C03656=1147.991,39.631,-50.274,-179.877,6.308,149.107
C03657=1147.986,39.881,-50.290,-179.875,6.309,149.107
C03658=1147.981,40.130,-50.305,-179.871,6.310,149.106
C03659=1147.976,40.380,-50.321,-179.869,6.311,149.106
C03660=1147.971,40.630,-50.335,-179.866,6.312,149.105
C03661=1147.966,40.879,-50.350,-179.864,6.313,149.105
C03662=1147.961,41.128,-50.365,-179.861,6.315,149.104
C03663=1147.956,41.378,-50.381,-179.859,6.315,149.104
C03664=1147.951,41.627,-50.395,-179.856,6.316,149.103
C03665=1147.945,41.877,-50.411,-179.853,6.317,149.102
C03666=1147.941,42.126,-50.426,-179.851,6.318,149.102
C03667=1147.936,42.376,-50.442,-179.848,6.320,149.102
C03668=1147.931,42.626,-50.456,-179.846,6.320,149.101
C03669=1147.926,42.875,-50.472,-179.843,6.322,149.100
C03670=1147.921,43.124,-50.487,-179.840,6.323,149.100
C03671=1147.916,43.374,-50.502,-179.838,6.323,149.099
C03672=1147.910,43.623,-50.518,-179.835,6.325,149.099
C03673=1147.906,43.872,-50.533,-179.833,6.325,149.098
C03674=1147.901,44.122,-50.549,-179.830,6.327,149.098
C03675=1147.896,44.372,-50.563,-179.827,6.328,149.097
C03676=1147.890,44.621,-50.579,-179.824,6.329,149.097
C03677=1147.885,44.871,-50.594,-179.822,6.330,149.096
C03678=1147.880,45.120,-50.609,-179.819,6.331,149.096
C03679=1147.876,45.370,-50.625,-179.817,6.332,149.095
C03680=1147.870,45.619,-50.641,-179.814,6.333,149.094
C03681=1147.866,45.868,-50.656,-179.812,6.334,149.094
C03682=1147.860,46.118,-50.671,-179.809,6.335,149.094
C03683=1147.856,46.367,-50.686,-179.806,6.336,149.093
C03684=1147.851,46.617,-50.702,-179.804,6.337,149.092
C03685=1147.845,46.866,-50.718,-179.801,6.339,149.092
C03686=1147.841,47.115,-50.733,-179.799,6.339,149.091
C03687=1147.835,47.365,-50.748,-179.796,6.341,149.091
C03688=1147.831,47.615,-50.764,-179.793,6.342,149.090
C03689=1147.826,47.864,-50.779,-179.790,6.343,149.090
C03690=1147.821,48.113,-50.795,-179.788,6.344,149.089
C03691=1147.815,48.363,-50.811,-179.785,6.345,149.089
C03692=1147.810,48.613,-50.827,-179.783,6.346,149.088
C03693=1147.806,48.862,-50.842,-179.780,6.347,149.088
C03694=1147.800,49.111,-50.857,-179.777,6.348,149.087
C03695=1147.795,49.361,-50.873,-179.775,6.349,149.087
C03696=1147.791,49.611,-50.888,-179.772,6.350,149.086
C03697=1147.785,49.860,-50.904,-179.770,6.351,149.086
C03698=1147.780,50.109,-50.919,-179.767,6.352,149.085
C03699=1147.775,50.359,-50.935,-179.765,6.353,149.084
C03700=1147.771,50.609,-50.950,-179.762,6.355,149.084
C03701=1147.765,50.858,-50.966,-179.759,6.355,149.083
C03702=1147.760,51.107,-50.982,-179.756,6.357,149.083
C03703=1147.755,51.357,-50.998,-179.754,6.358,149.082
C03704=1147.750,51.606,-51.014,-179.751,6.359,149.082
C03705=1147.745,51.855,-51.029,-179.749,6.360,149.081
C03706=1147.741,52.105,-51.045,-179.746,6.361,149.081
C03707=1147.735,52.355,-51.060,-179.743,6.362,149.080
C03708=1147.730,52.604,-51.076,-179.741,6.364,149.080
C03709=1147.725,52.854,-51.092,-179.738,6.364,149.079
C03710=1147.721,53.103,-51.107,-179.735,6.366,149.079
C03711=1147.715,53.371,-51.124,-179.732,6.367,149.078
C03712=1147.710,53.640,-51.141,-179.730,6.368,149.078
C03713=1147.704,53.908,-51.158,-179.727,6.369,149.077
C03714=1147.699,54.177,-51.176,-179.724,6.371,149.076
C03715=1147.694,54.427,-51.191,-179.721,6.371,149.076
C03716=1147.688,54.676,-51.207,-179.719,6.373,149.075
C03717=1147.684,54.926,-51.224,-179.716,6.374,149.075
C03718=1147.678,55.175,-51.239,-179.713,6.375,149.074
C03719=1147.673,55.425,-51.255,-179.711,6.376,149.074
C03720=1147.669,55.674,-51.270,-179.708,6.378,149.073
C03721=1147.664,55.923,-51.287,-179.706,6.378,149.073
C03722=1147.659,56.173,-51.302,-179.703,6.380,149.072
C03723=1147.654,56.423,-51.318,-179.700,6.380,149.072
C03724=1147.649,56.671,-51.334,-179.697,6.382,149.071
C03725=1147.644,56.922,-51.350,-179.695,6.383,149.071
C03726=1147.638,57.171,-51.366,-179.692,6.384,149.070
C03727=1147.633,57.420,-51.382,-179.689,6.386,149.070
C03728=1147.629,57.670,-51.398,-179.687,6.387,149.069
C03729=1147.624,57.919,-51.414,-179.684,6.388,149.068
C03730=1147.619,58.169,-51.430,-179.682,6.389,149.068
C03731=1147.613,58.418,-51.446,-179.679,6.390,149.068
C03732=1147.609,58.668,-51.463,-179.676,6.391,149.067
C03733=1147.603,58.917,-51.478,-179.674,6.393,149.067
C03734=1147.598,59.166,-51.495,-179.671,6.393,149.066
C03735=1147.594,59.416,-51.511,-179.668,6.395,149.065
C03736=1147.589,59.665,-51.527,-179.666,6.396,149.065
C03737=1147.584,59.915,-51.543,-179.663,6.397,149.064
C03738=1147.579,60.164,-51.559,-179.660,6.399,149.064
C03739=1147.574,60.414,-51.575,-179.658,6.399,149.063
C03740=1147.569,60.662,-51.591,-179.655,6.401,149.063
C03741=1147.564,60.913,-51.607,-179.653,6.402,149.062
C03742=1147.559,61.161,-51.624,-179.650,6.403,149.062
C03743=1147.554,61.411,-51.640,-179.647,6.404,149.061
C03744=1147.549,61.660,-51.656,-179.644,6.405,149.061
C03745=1147.544,61.910,-51.672,-179.642,6.406,149.060
C03746=1147.539,62.159,-51.688,-179.639,6.407,149.060
C03747=1147.534,62.409,-51.704,-179.636,6.409,149.059
C03748=1147.529,62.658,-51.720,-179.634,6.410,149.059
C03749=1147.524,62.908,-51.738,-179.631,6.411,149.058
C03750=1147.519,63.157,-51.753,-179.629,6.412,149.058
C03751=1147.514,63.407,-51.770,-179.626,6.414,149.057
C03752=1147.509,63.656,-51.785,-179.623,6.414,149.057
C03753=1147.504,63.906,-51.802,-179.621,6.416,149.056
C03754=1147.499,64.154,-51.818,-179.618,6.418,149.056
C03755=1147.495,64.404,-51.834,-179.615,6.418,149.055
C03756=1147.489,64.653,-51.851,-179.613,6.420,149.055
C03757=1147.484,64.903,-51.868,-179.610,6.420,149.054
C03758=1147.479,65.152,-51.884,-179.607,6.422,149.054
C03759=1147.474,65.402,-51.900,-179.604,6.424,149.053
C03760=1147.469,65.651,-51.917,-179.602,6.424,149.052
C03761=1147.464,65.901,-51.933,-179.599,6.426,149.052
C03762=1147.460,66.150,-51.949,-179.597,6.427,149.052
C03763=1147.454,66.399,-51.966,-179.594,6.428,149.051
C03764=1147.450,66.649,-51.983,-179.591,6.429,149.050
C03765=1147.444,66.898,-51.998,-179.589,6.430,149.050
C03766=1147.440,67.148,-52.015,-179.586,6.432,149.049
C03767=1147.435,67.397,-52.031,-179.583,6.432,149.049
C03768=1147.430,67.646,-52.049,-179.581,6.434,149.049
C03769=1147.425,67.896,-52.065,-179.577,6.435,149.048
C03770=1147.420,68.145,-52.081,-179.575,6.436,149.047
C03771=1147.415,68.395,-52.097,-179.572,6.438,149.047
C03772=1147.409,68.644,-52.114,-179.570,6.439,149.047
C03773=1147.405,68.893,-52.131,-179.567,6.440,149.046
C03774=1147.400,69.143,-52.148,-179.564,6.442,149.045
C03775=1147.395,69.392,-52.163,-179.562,6.443,149.045
C03776=1147.390,69.642,-52.181,-179.559,6.444,149.044
C03777=1147.385,69.891,-52.197,-179.556,6.446,149.044
C03778=1147.380,70.140,-52.214,-179.554,6.446,149.044
C03779=1147.375,70.390,-52.231,-179.551,6.448,149.043
C03780=1147.371,70.640,-52.247,-179.549,6.449,149.042
C03781=1147.365,70.888,-52.264,-179.546,6.450,149.042
C03782=1147.361,71.138,-52.280,-179.543,6.452,149.041
C03783=1147.355,71.387,-52.297,-179.541,6.452,149.041
C03784=1147.350,71.637,-52.313,-179.538,6.454,149.040
C03785=1147.346,71.886,-52.330,-179.535,6.455,149.040
C03786=1147.340,72.136,-52.347,-179.532,6.456,149.039
C03787=1147.336,72.385,-52.364,-179.530,6.458,149.039
C03788=1147.330,72.635,-52.381,-179.527,6.459,149.038
C03789=1147.326,72.884,-52.397,-179.524,6.460,149.038
C03790=1147.321,73.133,-52.414,-179.522,6.462,149.037
C03791=1147.316,73.383,-52.431,-179.519,6.463,149.037
C03792=1147.311,73.632,-52.448,-179.516,6.464,149.036
C03793=1147.306,73.881,-52.464,-179.514,6.466,149.036
C03794=1147.301,74.131,-52.481,-179.511,6.466,149.035
C03795=1147.296,74.380,-52.498,-179.508,6.468,149.035
C03796=1147.291,74.629,-52.516,-179.505,6.469,149.034
C03797=1147.286,74.878,-52.532,-179.503,6.470,149.034
C03798=1147.281,75.128,-52.550,-179.500,6.472,149.033
C03799=1147.277,75.378,-52.566,-179.497,6.473,149.033
C03800=1147.272,75.626,-52.582,-179.495,6.474,149.032
C03801=1147.266,75.876,-52.600,-179.492,6.475,149.032
C03802=1147.262,76.126,-52.616,-179.489,6.477,149.031
C03803=1147.257,76.376,-52.634,-179.487,6.478,149.031
C03804=1147.252,76.624,-52.650,-179.484,6.480,149.031
C03805=1147.246,76.874,-52.667,-179.481,6.481,149.030
C03806=1147.242,77.123,-52.685,-179.479,6.482,149.029
C03807=1147.237,77.373,-52.702,-179.476,6.483,149.029
C03808=1147.232,77.622,-52.718,-179.473,6.485,149.028
C03809=1147.227,77.871,-52.735,-179.471,6.486,149.028
C03810=1147.222,78.121,-52.752,-179.468,6.487,149.027
C03811=1147.217,78.370,-52.770,-179.465,6.489,149.027
C03812=1147.213,78.620,-52.787,-179.462,6.490,149.026
C03813=1147.207,78.869,-52.804,-179.460,6.491,149.026
C03814=1147.202,79.118,-52.821,-179.457,6.493,149.026
C03815=1147.197,79.387,-52.839,-179.454,6.494,149.025
C03816=1147.191,79.654,-52.858,-179.451,6.496,149.024
C03817=1147.187,79.923,-52.876,-179.448,6.497,149.024
C03818=1147.181,80.192,-52.895,-179.446,6.498,149.023
C03819=1147.176,80.441,-52.912,-179.443,6.499,149.023
C03820=1147.171,80.691,-52.928,-179.440,6.501,149.022
C03821=1147.166,80.940,-52.946,-179.437,6.502,149.022
C03822=1147.162,81.189,-52.963,-179.435,6.503,149.021
C03823=1147.156,81.439,-52.980,-179.432,6.505,149.021
C03824=1147.152,81.688,-52.998,-179.429,6.506,149.020
C03825=1147.147,81.938,-53.015,-179.427,6.507,149.020
C03826=1147.141,82.187,-53.032,-179.424,6.509,149.020
C03827=1147.136,82.436,-53.050,-179.421,6.510,149.019
C03828=1147.132,82.685,-53.067,-179.418,6.512,149.018
C03829=1147.127,82.935,-53.085,-179.416,6.513,149.018
C03830=1147.122,83.184,-53.102,-179.413,6.514,149.018
C03831=1147.117,83.434,-53.118,-179.410,6.516,149.017
C03832=1147.112,83.683,-53.136,-179.408,6.517,149.017
C03833=1147.107,83.933,-53.154,-179.405,6.518,149.016
C03834=1147.102,84.181,-53.171,-179.402,6.520,149.016
C03835=1147.097,84.431,-53.188,-179.399,6.521,149.015
C03836=1147.092,84.680,-53.206,-179.397,6.522,149.015
C03837=1147.088,84.929,-53.223,-179.394,6.524,149.014
C03838=1147.083,85.179,-53.241,-179.391,6.525,149.014
C03839=1147.078,85.428,-53.258,-179.388,6.527,149.013
C03840=1147.073,85.678,-53.276,-179.386,6.528,149.013
C03841=1147.068,85.927,-53.293,-179.384,6.529,149.012
C03842=1147.063,86.176,-53.311,-179.380,6.531,149.012
C03843=1147.058,86.426,-53.328,-179.378,6.532,149.011
C03844=1147.053,86.675,-53.346,-179.375,6.533,149.011
C03845=1147.049,86.925,-53.362,-179.373,6.535,149.010
C03846=1147.044,87.174,-53.380,-179.369,6.536,149.010
C03847=1147.038,87.422,-53.398,-179.367,6.538,149.009
C03848=1147.033,87.672,-53.415,-179.365,6.539,149.009
C03849=1147.028,87.921,-53.433,-179.362,6.540,149.008
C03850=1147.024,88.171,-53.450,-179.359,6.542,149.008
C03851=1147.019,88.420,-53.468,-179.356,6.543,149.007
C03852=1147.014,88.669,-53.486,-179.354,6.544,149.007
C03853=1147.009,88.919,-53.503,-179.351,6.546,149.007
C03854=1147.004,89.168,-53.521,-179.348,6.547,149.006
C03855=1147.000,89.417,-53.539,-179.345,6.549,149.005
C03856=1146.994,89.667,-53.556,-179.343,6.550,149.005
C03857=1146.989,89.916,-53.574,-179.340,6.551,149.005
C03858=1146.984,90.165,-53.592,-179.337,6.553,149.004
C03859=1146.979,90.415,-53.609,-179.334,6.554,149.004
C03860=1146.974,90.664,-53.627,-179.332,6.555,149.003
C03861=1146.969,90.913,-53.645,-179.329,6.557,149.003
C03862=1146.965,91.162,-53.663,-179.327,6.559,149.002
C03863=1146.960,91.412,-53.680,-179.323,6.560,149.002
C03864=1146.955,91.661,-53.698,-179.321,6.562,149.001
C03865=1146.951,91.911,-53.716,-179.319,6.562,149.001
C03866=1146.946,92.160,-53.734,-179.316,6.564,149.000
C03867=1146.941,92.410,-53.751,-179.313,6.565,149.000
C03868=1146.936,92.659,-53.769,-179.310,6.567,148.999
C03869=1146.931,92.908,-53.787,-179.308,6.568,148.999
C03870=1146.926,93.157,-53.805,-179.305,6.570,148.998
C03871=1146.921,93.407,-53.823,-179.302,6.571,148.998
C03872=1146.916,93.656,-53.840,-179.299,6.573,148.997
C03873=1146.911,93.906,-53.858,-179.296,6.574,148.997
C03874=1146.906,94.155,-53.876,-179.294,6.575,148.997
C03875=1146.901,94.404,-53.894,-179.291,6.577,148.996
C03876=1146.896,94.653,-53.912,-179.288,6.578,148.995
C03877=1146.891,94.902,-53.930,-179.285,6.580,148.995
C03878=1146.886,95.152,-53.948,-179.283,6.582,148.995
C03879=1146.882,95.401,-53.967,-179.281,6.582,148.994
C03880=1146.877,95.651,-53.985,-179.278,6.584,148.994
C03881=1146.872,95.900,-54.003,-179.275,6.585,148.993
C03882=1146.867,96.150,-54.020,-179.272,6.587,148.993
C03883=1146.862,96.399,-54.038,-179.269,6.589,148.992
C03884=1146.857,96.648,-54.056,-179.266,6.590,148.992
C03885=1146.852,96.897,-54.074,-179.264,6.591,148.991
C03886=1146.847,97.146,-54.092,-179.261,6.593,148.991
C03887=1146.843,97.396,-54.110,-179.258,6.594,148.990
C03888=1146.838,97.645,-54.128,-179.256,6.596,148.990
C03889=1146.833,97.894,-54.146,-179.253,6.598,148.990
C03890=1146.828,98.144,-54.164,-179.250,6.599,148.989
C03891=1146.823,98.393,-54.183,-179.248,6.600,148.989
C03892=1146.818,98.642,-54.201,-179.245,6.602,148.988
C03893=1146.814,98.892,-54.220,-179.242,6.603,148.988
C03894=1146.809,99.141,-54.238,-179.239,6.605,148.987
C03895=1146.804,99.390,-54.256,-179.237,6.607,148.987
C03896=1146.799,99.639,-54.274,-179.233,6.608,148.986
C03897=1146.794,99.888,-54.292,-179.231,6.609,148.986
C03898=1146.789,100.137,-54.310,-179.229,6.611,148.985
C03899=1146.784,100.388,-54.328,-179.226,6.612,148.985
C03900=1146.779,100.637,-54.346,-179.223,6.614,148.985
C03901=1146.774,100.886,-54.364,-179.220,6.615,148.984
C03902=1146.770,101.135,-54.383,-179.217,6.617,148.984
C03903=1146.765,101.384,-54.401,-179.215,6.618,148.983
C03904=1146.760,101.634,-54.419,-179.212,6.619,148.983
C03905=1146.755,101.883,-54.438,-179.210,6.621,148.982
C03906=1146.750,102.132,-54.456,-179.207,6.623,148.982
C03907=1146.745,102.381,-54.475,-179.204,6.624,148.981
C03908=1146.741,102.631,-54.493,-179.201,6.626,148.981
C03909=1146.735,102.880,-54.512,-179.198,6.628,148.980
C03910=1146.730,103.129,-54.530,-179.195,6.629,148.980
C03911=1146.726,103.378,-54.548,-179.193,6.630,148.980
C03912=1146.722,103.628,-54.567,-179.190,6.631,148.979
C03913=1146.716,103.877,-54.585,-179.187,6.633,148.979
C03914=1146.711,104.126,-54.603,-179.185,6.635,148.978
C03915=1146.707,104.376,-54.622,-179.182,6.636,148.978
C03916=1146.702,104.625,-54.640,-179.179,6.638,148.977
C03917=1146.696,104.874,-54.659,-179.176,6.640,148.977
C03918=1146.692,105.123,-54.678,-179.173,6.641,148.976
C03919=1146.687,105.392,-54.697,-179.170,6.643,148.976
C03920=1146.681,105.660,-54.717,-179.168,6.645,148.975
C03921=1146.676,105.929,-54.737,-179.165,6.646,148.975
C03922=1146.671,106.197,-54.757,-179.162,6.648,148.974
C03923=1146.667,106.447,-54.776,-179.159,6.649,148.974
C03924=1146.661,106.695,-54.795,-179.156,6.651,148.974
C03925=1146.656,106.945,-54.813,-179.154,6.653,148.973
C03926=1146.652,107.194,-54.831,-179.151,6.654,148.973
C03927=1146.647,107.443,-54.851,-179.148,6.655,148.972
C03928=1146.642,107.692,-54.869,-179.146,6.657,148.972
C03929=1146.638,107.942,-54.888,-179.143,6.658,148.971
C03930=1146.632,108.191,-54.906,-179.140,6.660,148.971
C03931=1146.628,108.440,-54.925,-179.137,6.662,148.970
C03932=1146.622,108.690,-54.944,-179.135,6.663,148.970
C03933=1146.618,108.939,-54.963,-179.132,6.665,148.970
C03934=1146.613,109.188,-54.981,-179.129,6.666,148.969
C03935=1146.608,109.437,-55.000,-179.126,6.668,148.969
C03936=1146.603,109.686,-55.018,-179.123,6.670,148.968
C03937=1146.598,109.935,-55.038,-179.121,6.671,148.968
C03938=1146.594,110.185,-55.056,-179.118,6.672,148.967
C03939=1146.588,110.434,-55.075,-179.116,6.674,148.967
C03940=1146.584,110.684,-55.094,-179.113,6.676,148.967
C03941=1146.579,110.933,-55.113,-179.110,6.677,148.966
C03942=1146.574,111.181,-55.132,-179.107,6.679,148.966
C03943=1146.569,111.432,-55.150,-179.104,6.680,148.965
C03944=1146.564,111.680,-55.169,-179.102,6.682,148.965
C03945=1146.559,111.930,-55.188,-179.099,6.684,148.964
C03946=1146.555,112.179,-55.207,-179.096,6.685,148.964
C03947=1146.550,112.428,-55.226,-179.093,6.687,148.963
C03948=1146.545,112.678,-55.244,-179.091,6.689,148.963
C03949=1146.540,112.926,-55.264,-179.087,6.690,148.962
C03950=1146.536,113.176,-55.283,-179.085,6.692,148.962
C03951=1146.530,113.425,-55.301,-179.082,6.693,148.962
C03952=1146.526,113.674,-55.320,-179.079,6.695,148.961
C03953=1146.521,113.923,-55.340,-179.077,6.696,148.961
C03954=1146.516,114.173,-55.358,-179.074,6.698,148.960
C03955=1146.511,114.422,-55.377,-179.072,6.699,148.960
C03956=1146.506,114.672,-55.397,-179.069,6.701,148.960
C03957=1146.502,114.920,-55.416,-179.066,6.703,148.959
C03958=1146.497,115.170,-55.435,-179.063,6.704,148.959
C03959=1146.492,115.419,-55.453,-179.060,6.706,148.958
C03960=1146.487,115.668,-55.473,-179.058,6.708,148.958
C03961=1146.482,115.917,-55.492,-179.055,6.709,148.957
C03962=1146.478,116.167,-55.511,-179.052,6.711,148.957
C03963=1146.472,116.416,-55.530,-179.049,6.713,148.957
C03964=1146.468,116.666,-55.550,-179.047,6.714,148.956
C03965=1146.463,116.914,-55.568,-179.044,6.716,148.956
C03966=1146.458,117.164,-55.588,-179.041,6.718,148.955
C03967=1146.453,117.413,-55.607,-179.038,6.719,148.955
C03968=1146.449,117.662,-55.626,-179.035,6.721,148.954
C03969=1146.444,117.911,-55.646,-179.033,6.722,148.954
C03970=1146.439,118.160,-55.665,-179.030,6.724,148.953
C03971=1146.434,118.410,-55.683,-179.027,6.726,148.953
C03972=1146.429,118.659,-55.703,-179.024,6.728,148.953
C03973=1146.424,118.908,-55.722,-179.022,6.729,148.952
C03974=1146.420,119.157,-55.741,-179.019,6.731,148.952
C03975=1146.415,119.407,-55.761,-179.016,6.733,148.951
C03976=1146.410,119.656,-55.780,-179.014,6.734,148.951
C03977=1146.405,119.905,-55.800,-179.011,6.736,148.951
C03978=1146.400,120.154,-55.818,-179.008,6.738,148.950
C03979=1146.396,120.403,-55.838,-179.005,6.739,148.950
C03980=1146.390,120.652,-55.857,-179.002,6.741,148.949
C03981=1146.386,120.902,-55.877,-178.999,6.742,148.949
C03982=1146.382,121.151,-55.896,-178.997,6.744,148.948
C03983=1146.376,121.400,-55.915,-178.994,6.746,148.948
C03984=1146.371,121.649,-55.935,-178.991,6.748,148.948
C03985=1146.366,121.898,-55.954,-178.989,6.749,148.947
C03986=1146.361,122.148,-55.974,-178.986,6.751,148.947
C03987=1146.357,122.397,-55.993,-178.983,6.753,148.946
C03988=1146.352,122.645,-56.013,-178.980,6.754,148.946
C03989=1146.348,122.895,-56.033,-178.978,6.756,148.946
C03990=1146.343,123.145,-56.052,-178.975,6.758,148.945
C03991=1146.337,123.393,-56.072,-178.972,6.759,148.945
C03992=1146.333,123.643,-56.091,-178.969,6.761,148.944
C03993=1146.329,123.892,-56.110,-178.967,6.763,148.944
C03994=1146.323,124.141,-56.130,-178.964,6.765,148.944
C03995=1146.319,124.390,-56.150,-178.961,6.766,148.943
C03996=1146.314,124.640,-56.170,-178.958,6.768,148.943
C03997=1146.309,124.889,-56.189,-178.955,6.769,148.942
C03998=1146.304,125.138,-56.209,-178.953,6.771,148.942
C03999=1146.299,125.388,-56.228,-178.950,6.773,148.941
C04000=1146.294,125.636,-56.248,-178.947,6.774,148.941
C04001=1146.290,125.885,-56.267,-178.945,6.776,148.941
C04002=1146.286,126.135,-56.287,-178.942,6.778,148.940
C04003=1146.280,126.384,-56.306,-178.939,6.780,148.940
C04004=1146.276,126.633,-56.327,-178.936,6.781,148.939
C04005=1146.271,126.882,-56.346,-178.934,6.783,148.939
C04006=1146.266,127.132,-56.366,-178.931,6.785,148.939
C04007=1146.261,127.380,-56.386,-178.928,6.786,148.938
C04008=1146.257,127.629,-56.406,-178.925,6.788,148.938
C04009=1146.252,127.879,-56.425,-178.922,6.791,148.937
C04010=1146.247,128.128,-56.446,-178.919,6.792,148.937
C04011=1146.242,128.377,-56.465,-178.917,6.794,148.937
C04012=1146.237,128.626,-56.485,-178.914,6.796,148.936
C04013=1146.233,128.875,-56.505,-178.911,6.797,148.936
C04014=1146.228,129.125,-56.525,-178.909,6.799,148.935
C04015=1146.223,129.374,-56.544,-178.906,6.801,148.935
C04016=1146.218,129.623,-56.564,-178.903,6.802,148.935
C04017=1146.214,129.872,-56.584,-178.900,6.804,148.934
C04018=1146.209,130.121,-56.604,-178.898,6.806,148.934
C04019=1146.204,130.370,-56.624,-178.895,6.808,148.933
C04020=1146.199,130.619,-56.644,-178.892,6.809,148.933
C04021=1146.195,130.869,-56.664,-178.890,6.811,148.933
C04022=1146.189,131.118,-56.685,-178.887,6.813,148.932
C04023=1146.185,131.387,-56.706,-178.884,6.815,148.932
C04024=1146.180,131.655,-56.727,-178.880,6.817,148.931
C04025=1146.174,131.924,-56.749,-178.878,6.818,148.931
C04026=1146.169,132.192,-56.770,-178.874,6.821,148.931
C04027=1146.164,132.441,-56.790,-178.872,6.822,148.930
C04028=1146.159,132.690,-56.811,-178.869,6.824,148.930
C04029=1146.154,132.939,-56.831,-178.866,6.826,148.929
C04030=1146.150,133.189,-56.851,-178.863,6.828,148.929
C04031=1146.145,133.438,-56.871,-178.861,6.829,148.929
C04032=1146.140,133.687,-56.891,-178.858,6.831,148.928
C04033=1146.136,133.936,-56.911,-178.855,6.833,148.928
C04034=1146.130,134.186,-56.931,-178.853,6.834,148.927
C04035=1146.125,134.434,-56.951,-178.849,6.837,148.927
C04036=1146.121,134.683,-56.972,-178.847,6.839,148.927
C04037=1146.116,134.933,-56.991,-178.844,6.840,148.926
C04038=1146.112,135.182,-57.012,-178.841,6.842,148.926
C04039=1146.107,135.431,-57.033,-178.838,6.844,148.925
C04040=1146.102,135.681,-57.052,-178.836,6.845,148.925
C04041=1146.098,135.930,-57.073,-178.833,6.847,148.925
C04042=1146.092,136.178,-57.093,-178.830,6.849,148.924
C04043=1146.088,136.427,-57.113,-178.828,6.851,148.924
C04044=1146.083,136.677,-57.133,-178.824,6.853,148.923
C04045=1146.078,136.926,-57.154,-178.822,6.855,148.923
C04046=1146.074,137.175,-57.174,-178.819,6.857,148.923
C04047=1146.069,137.424,-57.195,-178.816,6.858,148.922
C04048=1146.064,137.674,-57.215,-178.813,6.860,148.922
C04049=1146.059,137.922,-57.235,-178.811,6.862,148.922
C04050=1146.055,138.171,-57.255,-178.808,6.863,148.921
C04051=1146.050,138.421,-57.276,-178.805,6.866,148.921
C04052=1146.045,138.670,-57.297,-178.802,6.868,148.921
C04053=1146.041,138.919,-57.316,-178.800,6.870,148.920
C04054=1146.035,139.168,-57.337,-178.797,6.871,148.920
C04055=1146.031,139.417,-57.358,-178.794,6.873,148.919
C04056=1146.026,139.666,-57.378,-178.792,6.875,148.919
C04057=1146.021,139.916,-57.399,-178.789,6.876,148.919
C04058=1146.016,140.164,-57.419,-178.786,6.879,148.918
C04059=1146.012,140.413,-57.439,-178.783,6.881,148.918
C04060=1146.007,140.662,-57.460,-178.780,6.882,148.917
C04061=1146.002,140.912,-57.480,-178.777,6.884,148.917
C04062=1145.997,141.161,-57.501,-178.775,6.886,148.917
C04063=1145.992,141.410,-57.521,-178.772,6.888,148.916
C04064=1145.988,141.659,-57.542,-178.769,6.889,148.916
C04065=1145.983,141.909,-57.563,-178.766,6.892,148.916
C04066=1145.979,142.158,-57.584,-178.763,6.893,148.915
C04067=1145.974,142.407,-57.604,-178.761,6.895,148.915
C04068=1145.969,142.656,-57.625,-178.758,6.897,148.914
C04069=1145.965,142.905,-57.645,-178.756,6.899,148.914
C04070=1145.960,143.154,-57.666,-178.753,6.901,148.914
C04071=1145.955,143.403,-57.687,-178.750,6.903,148.913
C04072=1145.950,143.652,-57.708,-178.747,6.905,148.913
C04073=1145.946,143.901,-57.729,-178.744,6.907,148.913
C04074=1145.941,144.150,-57.750,-178.741,6.908,148.912
C04075=1145.936,144.399,-57.770,-178.739,6.910,148.912
C04076=1145.931,144.648,-57.791,-178.735,6.913,148.912
C04077=1145.927,144.897,-57.811,-178.733,6.914,148.911
C04078=1145.922,145.146,-57.832,-178.730,6.916,148.911
C04079=1145.917,145.395,-57.853,-178.727,6.918,148.910
C04080=1145.912,145.645,-57.874,-178.725,6.919,148.910
C04081=1145.907,145.893,-57.894,-178.722,6.922,148.910
C04082=1145.903,146.143,-57.916,-178.719,6.924,148.909
C04083=1145.899,146.392,-57.936,-178.716,6.926,148.909
C04084=1145.894,146.641,-57.957,-178.714,6.927,148.909
C04085=1145.888,146.890,-57.978,-178.711,6.929,148.908
C04086=1145.884,147.139,-57.999,-178.708,6.931,148.908
C04087=1145.879,147.388,-58.020,-178.705,6.933,148.908
C04088=1145.875,147.637,-58.041,-178.702,6.935,148.907
C04089=1145.869,147.886,-58.062,-178.699,6.937,148.907
C04090=1145.865,148.136,-58.083,-178.697,6.939,148.906
C04091=1145.861,148.384,-58.104,-178.695,6.941,148.906
C04092=1145.856,148.634,-58.125,-178.691,6.943,148.906
C04093=1145.851,148.883,-58.145,-178.689,6.945,148.905
C04094=1145.846,149.131,-58.167,-178.686,6.947,148.905
C04095=1145.841,149.380,-58.188,-178.683,6.948,148.905
C04096=1145.837,149.629,-58.209,-178.680,6.951,148.904
C04097=1145.832,149.879,-58.230,-178.677,6.953,148.904
C04098=1145.827,150.128,-58.252,-178.674,6.954,148.904
C04099=1145.823,150.377,-58.272,-178.672,6.956,148.903
C04100=1145.818,150.626,-58.294,-178.669,6.958,148.903
C04101=1145.813,150.875,-58.315,-178.666,6.961,148.903
C04102=1145.808,151.125,-58.336,-178.663,6.962,148.902
C04103=1145.804,151.373,-58.357,-178.661,6.964,148.902
C04104=1145.799,151.622,-58.378,-178.658,6.966,148.901
C04105=1145.794,151.871,-58.400,-178.655,6.968,148.901
C04106=1145.790,152.120,-58.420,-178.652,6.970,148.901
C04107=1145.785,152.369,-58.442,-178.650,6.972,148.901
C04108=1145.780,152.619,-58.463,-178.647,6.974,148.900
C04109=1145.775,152.868,-58.484,-178.644,6.976,148.900
C04110=1145.770,153.117,-58.506,-178.641,6.978,148.899
C04111=1145.766,153.366,-58.526,-178.638,6.980,148.899
C04112=1145.761,153.615,-58.548,-178.636,6.981,148.899
C04113=1145.757,153.863,-58.570,-178.632,6.984,148.898
C04114=1145.751,154.113,-58.591,-178.630,6.986,148.898
C04115=1145.747,154.362,-58.613,-178.627,6.988,148.898
C04116=1145.743,154.611,-58.633,-178.625,6.990,148.897
C04117=1145.738,154.860,-58.655,-178.621,6.992,148.897
C04118=1145.733,155.109,-58.676,-178.619,6.994,148.897
C04119=1145.728,155.358,-58.698,-178.616,6.995,148.896
C04120=1145.723,155.607,-58.720,-178.614,6.998,148.896
C04121=1145.718,155.856,-58.740,-178.610,7.000,148.896
C04122=1145.715,156.105,-58.762,-178.608,7.002,148.895
C04123=1145.710,156.354,-58.783,-178.605,7.004,148.895
C04124=1145.705,156.603,-58.805,-178.602,7.006,148.895
C04125=1145.700,156.852,-58.826,-178.599,7.008,148.894
C04126=1145.695,157.102,-58.848,-178.597,7.010,148.894
C04127=1145.691,157.370,-58.871,-178.594,7.012,148.894
C04128=1145.685,157.639,-58.894,-178.591,7.014,148.893
C04129=1145.681,157.909,-58.917,-178.588,7.017,148.893
C04130=1145.675,158.177,-58.941,-178.585,7.018,148.893
C04131=1145.670,158.427,-58.962,-178.582,7.021,148.892
C04132=1145.665,158.675,-58.984,-178.579,7.023,148.892
C04133=1145.661,158.924,-59.006,-178.576,7.024,148.892
C04134=1145.656,159.173,-59.028,-178.574,7.026,148.891
C04135=1145.651,159.422,-59.049,-178.571,7.029,148.891
C04136=1145.647,159.672,-59.071,-178.568,7.031,148.891
C04137=1145.642,159.920,-59.092,-178.565,7.032,148.890
C04138=1145.637,160.169,-59.114,-178.562,7.035,148.890
C04139=1145.633,160.418,-59.136,-178.560,7.037,148.890
C04140=1145.628,160.667,-59.158,-178.557,7.039,148.889
C04141=1145.624,160.916,-59.180,-178.554,7.041,148.889
C04142=1145.618,161.166,-59.201,-178.551,7.043,148.889
C04143=1145.614,161.414,-59.222,-178.548,7.045,148.888
C04144=1145.609,161.664,-59.245,-178.545,7.048,148.888
C04145=1145.604,161.912,-59.266,-178.543,7.049,148.888
C04146=1145.600,162.162,-59.288,-178.540,7.051,148.887
C04147=1145.595,162.410,-59.310,-178.537,7.054,148.887
C04148=1145.591,162.660,-59.332,-178.534,7.055,148.887
C04149=1145.586,162.908,-59.354,-178.532,7.057,148.886
C04150=1145.581,163.157,-59.375,-178.529,7.059,148.886
C04151=1145.577,163.406,-59.397,-178.526,7.062,148.886
C04152=1145.572,163.655,-59.419,-178.523,7.063,148.885
C04153=1145.568,163.904,-59.441,-178.521,7.065,148.885
C04154=1145.562,164.153,-59.463,-178.518,7.068,148.885
C04155=1145.558,164.402,-59.485,-178.515,7.070,148.884
C04156=1145.553,164.651,-59.507,-178.512,7.071,148.884
C04157=1145.549,164.900,-59.529,-178.509,7.074,148.884
C04158=1145.544,165.149,-59.551,-178.507,7.076,148.884
C04159=1145.540,165.398,-59.573,-178.503,7.079,148.883
C04160=1145.535,165.647,-59.595,-178.501,7.080,148.883
C04161=1145.530,165.897,-59.617,-178.498,7.082,148.883
C04162=1145.525,166.145,-59.639,-178.495,7.085,148.882
C04163=1145.521,166.394,-59.662,-178.492,7.087,148.882
C04164=1145.516,166.643,-59.683,-178.490,7.088,148.882
C04165=1145.512,166.892,-59.705,-178.487,7.091,148.881
C04166=1145.506,167.141,-59.728,-178.484,7.093,148.881
C04167=1145.502,167.390,-59.750,-178.482,7.095,148.881
C04168=1145.497,167.639,-59.771,-178.478,7.097,148.880
C04169=1145.493,167.888,-59.794,-178.476,7.099,148.880
C04170=1145.488,168.137,-59.816,-178.473,7.101,148.880
C04171=1145.483,168.386,-59.839,-178.470,7.104,148.880
C04172=1145.479,168.635,-59.861,-178.467,7.105,148.879
C04173=1145.474,168.884,-59.882,-178.464,7.108,148.879
C04174=1145.469,169.133,-59.906,-178.462,7.110,148.879
C04175=1145.465,169.382,-59.927,-178.459,7.112,148.878
C04176=1145.460,169.631,-59.949,-178.456,7.114,148.878
C04177=1145.455,169.879,-59.972,-178.454,7.116,148.878
C04178=1145.451,170.129,-59.994,-178.451,7.118,148.877
C04179=1145.447,170.378,-60.016,-178.448,7.121,148.877
C04180=1145.441,170.626,-60.039,-178.445,7.123,148.877
C04181=1145.437,170.876,-60.061,-178.442,7.125,148.877
C04182=1145.432,171.124,-60.083,-178.439,7.127,148.876
C04183=1145.427,171.373,-60.106,-178.437,7.129,148.876
C04184=1145.423,171.623,-60.129,-178.434,7.132,148.876
C04185=1145.418,171.871,-60.150,-178.431,7.133,148.875
C04186=1145.414,172.120,-60.174,-178.428,7.136,148.875
C04187=1145.409,172.369,-60.195,-178.426,7.138,148.875
C04188=1145.404,172.618,-60.219,-178.423,7.140,148.874
C04189=1145.400,172.867,-60.241,-178.420,7.142,148.874
C04190=1145.395,173.116,-60.262,-178.417,7.144,148.874
C04191=1145.390,173.365,-60.286,-178.414,7.147,148.874
C04192=1145.386,173.614,-60.308,-178.411,7.149,148.873
C04193=1145.381,173.863,-60.331,-178.409,7.151,148.873
C04194=1145.376,174.112,-60.353,-178.406,7.153,148.873
C04195=1145.372,174.361,-60.376,-178.403,7.155,148.872
C04196=1145.367,174.610,-60.398,-178.400,7.157,148.872
C04197=1145.362,174.859,-60.421,-178.398,7.160,148.872
C04198=1145.358,175.107,-60.444,-178.395,7.161,148.871
C04199=1145.354,175.357,-60.466,-178.392,7.164,148.871
C04200=1145.349,175.605,-60.489,-178.390,7.166,148.871
C04201=1145.344,175.854,-60.511,-178.386,7.168,148.871
C04202=1145.340,176.104,-60.534,-178.384,7.170,148.870
C04203=1145.335,176.352,-60.556,-178.381,7.173,148.870
C04204=1145.330,176.601,-60.579,-178.378,7.175,148.870
C04205=1145.325,176.850,-60.603,-178.375,7.177,148.869
C04206=1145.321,177.100,-60.625,-178.373,7.179,148.869
C04207=1145.316,177.348,-60.648,-178.370,7.181,148.869
C04208=1145.312,177.597,-60.671,-178.367,7.184,148.869
C04209=1145.307,177.846,-60.693,-178.364,7.186,148.868
C04210=1145.303,178.095,-60.716,-178.361,7.188,148.868
C04211=1145.297,178.343,-60.739,-178.359,7.190,148.868
C04212=1145.294,178.592,-60.762,-178.356,7.193,148.868
C04213=1145.289,178.842,-60.784,-178.353,7.195,148.867
C04214=1145.284,179.091,-60.808,-178.351,7.197,148.867
C04215=1145.279,179.339,-60.830,-178.347,7.199,148.867
C04216=1145.275,179.588,-60.854,-178.345,7.201,148.866
C04217=1145.270,179.837,-60.876,-178.342,7.204,148.866
C04218=1145.266,180.086,-60.899,-178.339,7.206,148.866
C04219=1145.261,180.335,-60.922,-178.336,7.208,148.866
C04220=1145.256,180.583,-60.945,-178.334,7.210,148.865
C04221=1145.252,180.832,-60.968,-178.330,7.213,148.865
C04222=1145.247,181.082,-60.991,-178.328,7.215,148.865
C04223=1145.243,181.331,-61.013,-178.325,7.218,148.865
C04224=1145.238,181.580,-61.037,-178.322,7.219,148.864
C04225=1145.233,181.829,-61.060,-178.319,7.222,148.864
C04226=1145.229,182.077,-61.083,-178.317,7.224,148.864
C04227=1145.224,182.326,-61.106,-178.313,7.226,148.863
C04228=1145.219,182.575,-61.129,-178.311,7.229,148.863
C04229=1145.215,182.824,-61.153,-178.308,7.230,148.863
C04230=1145.211,183.073,-61.175,-178.306,7.233,148.863
C04231=1145.205,183.342,-61.200,-178.302,7.236,148.862
C04232=1145.200,183.612,-61.226,-178.299,7.238,148.862
C04233=1145.195,183.882,-61.251,-178.296,7.240,148.862
C04234=1145.190,184.151,-61.275,-178.294,7.243,148.862
C04235=1145.185,184.400,-61.298,-178.290,7.245,148.861
C04236=1145.181,184.649,-61.322,-178.288,7.248,148.861
C04237=1145.176,184.898,-61.346,-178.285,7.250,148.861
C04238=1145.172,185.147,-61.369,-178.282,7.252,148.860
C04239=1145.168,185.395,-61.392,-178.279,7.255,148.860
C04240=1145.163,185.645,-61.415,-178.277,7.256,148.860
C04241=1145.158,185.894,-61.439,-178.274,7.259,148.860
C04242=1145.154,186.143,-61.462,-178.271,7.261,148.859
C04243=1145.148,186.391,-61.485,-178.268,7.264,148.859
C04244=1145.144,186.640,-61.508,-178.266,7.266,148.859
C04245=1145.140,186.889,-61.531,-178.262,7.268,148.859
C04246=1145.135,187.138,-61.554,-178.260,7.270,148.859
C04247=1145.130,187.387,-61.578,-178.257,7.273,148.858
C04248=1145.126,187.635,-61.602,-178.255,7.275,148.858
C04249=1145.121,187.884,-61.625,-178.251,7.278,148.858
C04250=1145.116,188.133,-61.649,-178.249,7.280,148.858
C04251=1145.112,188.382,-61.672,-178.246,7.282,148.857
C04252=1145.107,188.631,-61.695,-178.243,7.284,148.857
C04253=1145.103,188.880,-61.719,-178.240,7.287,148.857
C04254=1145.098,189.129,-61.743,-178.238,7.289,148.856
C04255=1145.093,189.378,-61.766,-178.235,7.291,148.856
C04256=1145.088,189.627,-61.789,-178.232,7.293,148.856
C04257=1145.085,189.875,-61.813,-178.229,7.296,148.856
C04258=1145.080,190.124,-61.836,-178.227,7.298,148.855
C04259=1145.075,190.373,-61.860,-178.224,7.301,148.855
C04260=1145.071,190.621,-61.884,-178.221,7.303,148.855
C04261=1145.066,190.870,-61.907,-178.218,7.305,148.855
C04262=1145.062,191.119,-61.930,-178.215,7.308,148.855
C04263=1145.057,191.368,-61.955,-178.212,7.310,148.854
C04264=1145.052,191.617,-61.978,-178.210,7.313,148.854
C04265=1145.047,191.866,-62.002,-178.207,7.314,148.854
C04266=1145.043,192.115,-62.026,-178.204,7.317,148.854
C04267=1145.038,192.364,-62.049,-178.201,7.319,148.853
C04268=1145.034,192.612,-62.073,-178.199,7.322,148.853
C04269=1145.029,192.861,-62.097,-178.195,7.324,148.853
C04270=1145.024,193.110,-62.120,-178.193,7.327,148.853
C04271=1145.020,193.359,-62.144,-178.190,7.329,148.852
C04272=1145.015,193.608,-62.167,-178.188,7.331,148.852
C04273=1145.011,193.857,-62.192,-178.184,7.334,148.852
C04274=1145.007,194.106,-62.215,-178.182,7.336,148.852
C04275=1145.002,194.354,-62.239,-178.179,7.338,148.851
C04276=1144.998,194.603,-62.263,-178.176,7.341,148.851
C04277=1144.992,194.852,-62.287,-178.173,7.343,148.851
C04278=1144.988,195.101,-62.311,-178.170,7.346,148.851
C04279=1144.983,195.349,-62.335,-178.168,7.348,148.850
C04280=1144.979,195.598,-62.359,-178.165,7.351,148.850
C04281=1144.974,195.847,-62.382,-178.162,7.352,148.850
C04282=1144.970,196.096,-62.407,-178.159,7.355,148.850
C04283=1144.965,196.345,-62.431,-178.156,7.358,148.850
C04284=1144.961,196.594,-62.455,-178.154,7.360,148.849
C04285=1144.956,196.842,-62.479,-178.151,7.362,148.849
C04286=1144.951,197.091,-62.502,-178.148,7.365,148.849
C04287=1144.947,197.340,-62.526,-178.145,7.367,148.849
C04288=1144.942,197.588,-62.551,-178.142,7.370,148.848
C04289=1144.938,197.838,-62.575,-178.140,7.372,148.848
C04290=1144.933,198.086,-62.599,-178.137,7.375,148.848
C04291=1144.929,198.335,-62.623,-178.135,7.377,148.848
C04292=1144.924,198.584,-62.647,-178.131,7.379,148.848
C04293=1144.919,198.833,-62.671,-178.129,7.382,148.847
C04294=1144.915,199.082,-62.695,-178.126,7.384,148.847
C04295=1144.911,199.330,-62.719,-178.123,7.387,148.847
C04296=1144.906,199.579,-62.743,-178.120,7.389,148.847
C04297=1144.901,199.828,-62.767,-178.118,7.391,148.847
C04298=1144.897,200.076,-62.791,-178.114,7.394,148.846
C04299=1144.892,200.326,-62.816,-178.112,7.396,148.846
C04300=1144.888,200.574,-62.841,-178.109,7.399,148.846
C04301=1144.883,200.823,-62.864,-178.107,7.401,148.846
C04302=1144.879,201.072,-62.888,-178.104,7.404,148.845
C04303=1144.874,201.321,-62.913,-178.101,7.406,148.845
C04304=1144.870,201.569,-62.937,-178.098,7.408,148.845
C04305=1144.865,201.818,-62.962,-178.095,7.411,148.845
C04306=1144.860,202.066,-62.986,-178.092,7.414,148.845
C04307=1144.857,202.316,-63.010,-178.090,7.416,148.844
C04308=1144.851,202.564,-63.035,-178.087,7.418,148.844
C04309=1144.847,202.813,-63.059,-178.084,7.421,148.844
C04310=1144.842,203.062,-63.082,-178.081,7.423,148.844
C04311=1144.838,203.311,-63.107,-178.078,7.426,148.844
C04312=1144.833,203.560,-63.131,-178.076,7.428,148.843
C04313=1144.828,203.808,-63.156,-178.073,7.431,148.843
C04314=1144.824,204.057,-63.181,-178.070,7.434,148.843
C04315=1144.819,204.306,-63.205,-178.067,7.435,148.843
C04316=1144.815,204.555,-63.229,-178.065,7.438,148.843
C04317=1144.810,204.804,-63.254,-178.061,7.441,148.842
C04318=1144.806,205.052,-63.279,-178.059,7.443,148.842
C04319=1144.802,205.300,-63.303,-178.056,7.446,148.842
C04320=1144.797,205.550,-63.328,-178.053,7.448,148.842
C04321=1144.792,205.798,-63.353,-178.051,7.450,148.842
C04322=1144.788,206.047,-63.377,-178.048,7.453,148.841
C04323=1144.783,206.296,-63.402,-178.045,7.456,148.841
C04324=1144.779,206.545,-63.426,-178.043,7.458,148.841
C04325=1144.774,206.793,-63.451,-178.039,7.461,148.841
C04326=1144.770,207.042,-63.475,-178.037,7.463,148.841
C04327=1144.765,207.291,-63.500,-178.034,7.466,148.840
C04328=1144.761,207.539,-63.525,-178.031,7.468,148.840
C04329=1144.756,207.788,-63.550,-178.028,7.471,148.840
C04330=1144.752,208.037,-63.574,-178.026,7.473,148.840
C04331=1144.747,208.286,-63.599,-178.023,7.476,148.840
C04332=1144.742,208.535,-63.624,-178.020,7.479,148.839
C04333=1144.738,208.783,-63.648,-178.017,7.480,148.839
C04334=1144.734,209.032,-63.673,-178.014,7.483,148.839
C04335=1144.728,209.302,-63.700,-178.012,7.486,148.839
C04336=1144.724,209.573,-63.727,-178.008,7.489,148.839
C04337=1144.719,209.843,-63.754,-178.006,7.492,148.839
C04338=1144.714,210.114,-63.781,-178.002,7.494,148.838
C04339=1144.709,210.363,-63.806,-178.000,7.497,148.838
C04340=1144.705,210.612,-63.831,-177.997,7.500,148.838
C04341=1144.700,210.860,-63.855,-177.994,7.502,148.838
C04342=1144.696,211.110,-63.880,-177.991,7.505,148.838
C04343=1144.691,211.358,-63.906,-177.988,7.508,148.837
C04344=1144.687,211.607,-63.930,-177.986,7.509,148.837
C04345=1144.682,211.855,-63.956,-177.983,7.512,148.837
C04346=1144.677,212.104,-63.980,-177.980,7.515,148.837
C04347=1144.673,212.353,-64.005,-177.977,7.518,148.837
C04348=1144.669,212.601,-64.030,-177.975,7.520,148.836
C04349=1144.664,212.850,-64.055,-177.972,7.523,148.836
C04350=1144.659,213.098,-64.081,-177.969,7.525,148.836
C04351=1144.655,213.348,-64.106,-177.966,7.527,148.836
C04352=1144.651,213.596,-64.130,-177.964,7.530,148.836
C04353=1144.646,213.845,-64.155,-177.960,7.533,148.836
C04354=1144.641,214.093,-64.181,-177.958,7.536,148.835
C04355=1144.637,214.343,-64.206,-177.955,7.538,148.835
C04356=1144.633,214.591,-64.231,-177.952,7.540,148.835
C04357=1144.628,214.840,-64.256,-177.949,7.543,148.835
C04358=1144.624,215.089,-64.281,-177.946,7.546,148.835
C04359=1144.619,215.337,-64.306,-177.944,7.548,148.835
C04360=1144.615,215.586,-64.332,-177.941,7.551,148.834
C04361=1144.610,215.834,-64.357,-177.938,7.554,148.834
C04362=1144.606,216.083,-64.382,-177.935,7.557,148.834
C04363=1144.601,216.331,-64.407,-177.933,7.559,148.834
C04364=1144.597,216.580,-64.433,-177.930,7.561,148.834
C04365=1144.592,216.830,-64.458,-177.927,7.564,148.834
C04366=1144.588,217.078,-64.483,-177.924,7.567,148.834
C04367=1144.583,217.327,-64.509,-177.922,7.569,148.833
C04368=1144.578,217.575,-64.534,-177.919,7.572,148.833
C04369=1144.574,217.824,-64.559,-177.916,7.575,148.833
C04370=1144.571,218.073,-64.585,-177.913,7.578,148.833
C04371=1144.565,218.321,-64.609,-177.911,7.580,148.833
C04372=1144.561,218.570,-64.635,-177.908,7.582,148.832
C04373=1144.556,218.818,-64.660,-177.905,7.585,148.832
C04374=1144.552,219.067,-64.686,-177.902,7.588,148.832
C04375=1144.548,219.316,-64.712,-177.899,7.590,148.832
C04376=1144.543,219.565,-64.737,-177.897,7.593,148.832
C04377=1144.539,219.813,-64.762,-177.894,7.596,148.832
C04378=1144.534,220.062,-64.788,-177.891,7.599,148.832
C04379=1144.530,220.310,-64.813,-177.888,7.601,148.831
C04380=1144.525,220.559,-64.839,-177.886,7.603,148.831
C04381=1144.521,220.808,-64.865,-177.883,7.606,148.831
C04382=1144.516,221.057,-64.890,-177.880,7.609,148.831
C04383=1144.512,221.305,-64.915,-177.877,7.612,148.831
C04384=1144.508,221.554,-64.941,-177.875,7.614,148.831
C04385=1144.503,221.802,-64.966,-177.872,7.617,148.831
C04386=1144.498,222.051,-64.992,-177.869,7.620,148.830
C04387=1144.494,222.300,-65.018,-177.866,7.622,148.830
C04388=1144.489,222.548,-65.043,-177.863,7.625,148.830
C04389=1144.484,222.797,-65.070,-177.861,7.627,148.830
C04390=1144.480,223.046,-65.095,-177.858,7.630,148.830
C04391=1144.475,223.294,-65.121,-177.855,7.633,148.830
C04392=1144.471,223.543,-65.147,-177.852,7.636,148.829
C04393=1144.467,223.792,-65.172,-177.849,7.639,148.829
C04394=1144.463,224.041,-65.198,-177.847,7.641,148.829
C04395=1144.458,224.289,-65.223,-177.844,7.644,148.829
C04396=1144.454,224.537,-65.249,-177.841,7.647,148.829
C04397=1144.449,224.786,-65.275,-177.838,7.649,148.829
C04398=1144.444,225.035,-65.301,-177.835,7.652,148.829
C04399=1144.440,225.283,-65.327,-177.833,7.654,148.828
C04400=1144.436,225.532,-65.353,-177.830,7.657,148.828
C04401=1144.432,225.780,-65.379,-177.827,7.660,148.828
C04402=1144.427,226.029,-65.405,-177.824,7.663,148.828
C04403=1144.422,226.278,-65.431,-177.821,7.666,148.828
C04404=1144.417,226.526,-65.456,-177.818,7.668,148.828
C04405=1144.413,226.775,-65.482,-177.816,7.671,148.828
C04406=1144.409,227.024,-65.508,-177.813,7.673,148.828
C04407=1144.405,227.272,-65.534,-177.810,7.676,148.827
C04408=1144.400,227.521,-65.560,-177.807,7.679,148.827
C04409=1144.395,227.769,-65.586,-177.805,7.682,148.827
C04410=1144.391,228.018,-65.612,-177.802,7.685,148.827
C04411=1144.386,228.267,-65.639,-177.800,7.687,148.827
C04412=1144.382,228.516,-65.665,-177.797,7.690,148.827
C04413=1144.377,228.764,-65.690,-177.794,7.692,148.827
C04414=1144.373,229.012,-65.717,-177.791,7.695,148.826
C04415=1144.369,229.261,-65.743,-177.788,7.698,148.826
C04416=1144.364,229.510,-65.769,-177.785,7.701,148.826
C04417=1144.360,229.759,-65.794,-177.783,7.703,148.826
C04418=1144.355,230.007,-65.821,-177.780,7.706,148.826
C04419=1144.351,230.256,-65.847,-177.777,7.709,148.826
C04420=1144.347,230.503,-65.873,-177.774,7.712,148.826
C04421=1144.342,230.752,-65.900,-177.771,7.715,148.826
C04422=1144.337,231.001,-65.925,-177.769,7.717,148.826
C04423=1144.334,231.249,-65.952,-177.766,7.720,148.825
C04424=1144.329,231.499,-65.978,-177.764,7.722,148.825
C04425=1144.325,231.747,-66.005,-177.761,7.725,148.825
C04426=1144.320,231.996,-66.031,-177.758,7.728,148.825
C04427=1144.316,232.244,-66.057,-177.755,7.731,148.825
C04428=1144.312,232.493,-66.083,-177.752,7.734,148.825
C04429=1144.306,232.741,-66.110,-177.749,7.737,148.825
C04430=1144.302,232.989,-66.136,-177.746,7.740,148.825
C04431=1144.297,233.238,-66.163,-177.743,7.743,148.825
C04432=1144.293,233.487,-66.188,-177.741,7.745,148.824
C04433=1144.289,233.735,-66.216,-177.738,7.748,148.824
C04434=1144.284,233.984,-66.241,-177.736,7.751,148.824
C04435=1144.280,234.233,-66.268,-177.733,7.753,148.824
C04436=1144.275,234.481,-66.294,-177.730,7.756,148.824
C04437=1144.271,234.730,-66.321,-177.727,7.759,148.824
C04438=1144.267,234.978,-66.348,-177.724,7.762,148.824
C04439=1144.261,235.250,-66.376,-177.721,7.765,148.824
C04440=1144.257,235.522,-66.405,-177.718,7.768,148.824
C04441=1144.253,235.794,-66.435,-177.716,7.771,148.823
C04442=1144.247,236.066,-66.463,-177.712,7.774,148.823
C04443=1144.243,236.314,-66.490,-177.709,7.777,148.823
C04444=1144.239,236.563,-66.517,-177.706,7.780,148.823
C04445=1144.234,236.811,-66.544,-177.704,7.782,148.823
C04446=1144.230,237.060,-66.570,-177.701,7.785,148.823
C04447=1144.225,237.309,-66.597,-177.698,7.788,148.823
C04448=1144.221,237.557,-66.623,-177.696,7.791,148.823
C04449=1144.216,237.805,-66.650,-177.693,7.794,148.823
C04450=1144.211,238.054,-66.677,-177.690,7.797,148.823
C04451=1144.208,238.303,-66.703,-177.687,7.799,148.822
C04452=1144.203,238.551,-66.730,-177.684,7.802,148.822
C04453=1144.199,238.799,-66.757,-177.682,7.805,148.822
C04454=1144.194,239.048,-66.784,-177.679,7.808,148.822
C04455=1144.189,239.297,-66.810,-177.676,7.811,148.822
C04456=1144.185,239.545,-66.837,-177.673,7.813,148.822
C04457=1144.181,239.793,-66.864,-177.671,7.816,148.822
C04458=1144.177,240.043,-66.891,-177.668,7.819,148.822
C04459=1144.173,240.291,-66.917,-177.665,7.822,148.822
C04460=1144.168,240.539,-66.945,-177.662,7.825,148.821
C04461=1144.163,240.788,-66.972,-177.659,7.827,148.821
C04462=1144.159,241.036,-66.999,-177.657,7.830,148.821
C04463=1144.155,241.285,-67.025,-177.654,7.833,148.821
C04464=1144.150,241.533,-67.052,-177.651,7.836,148.821
C04465=1144.146,241.782,-67.079,-177.648,7.839,148.821
C04466=1144.141,242.030,-67.106,-177.646,7.842,148.821
C04467=1144.137,242.278,-67.133,-177.643,7.845,148.821
C04468=1144.133,242.527,-67.160,-177.640,7.848,148.821
C04469=1144.128,242.776,-67.187,-177.637,7.851,148.821
C04470=1144.124,243.024,-67.214,-177.635,7.853,148.821
C04471=1144.120,243.273,-67.241,-177.632,7.856,148.821
C04472=1144.115,243.521,-67.268,-177.629,7.859,148.821
C04473=1144.110,243.770,-67.295,-177.627,7.862,148.820
C04474=1144.106,244.019,-67.322,-177.624,7.865,148.820
C04475=1144.102,244.267,-67.349,-177.621,7.868,148.820
C04476=1144.097,244.516,-67.376,-177.618,7.870,148.820
C04477=1144.093,244.763,-67.404,-177.615,7.873,148.820
C04478=1144.089,245.012,-67.431,-177.613,7.876,148.820
C04479=1144.084,245.260,-67.458,-177.610,7.879,148.820
C04480=1144.080,245.510,-67.485,-177.607,7.882,148.820
C04481=1144.075,245.758,-67.512,-177.604,7.885,148.820
C04482=1144.071,246.007,-67.539,-177.601,7.888,148.820
C04483=1144.066,246.254,-67.567,-177.599,7.891,148.820
C04484=1144.062,246.503,-67.594,-177.596,7.894,148.820
C04485=1144.058,246.752,-67.622,-177.593,7.897,148.820
C04486=1144.054,247.000,-67.648,-177.590,7.900,148.819
C04487=1144.049,247.248,-67.676,-177.587,7.903,148.819
C04488=1144.045,247.497,-67.703,-177.585,7.906,148.819
C04489=1144.041,247.746,-67.730,-177.582,7.908,148.819
C04490=1144.036,247.994,-67.758,-177.579,7.911,148.819
C04491=1144.032,248.242,-67.785,-177.576,7.914,148.819
C04492=1144.027,248.491,-67.812,-177.574,7.917,148.819
C04493=1144.023,248.739,-67.840,-177.571,7.920,148.819
C04494=1144.019,248.988,-67.867,-177.568,7.923,148.819
C04495=1144.014,249.236,-67.894,-177.565,7.926,148.819
C04496=1144.010,249.485,-67.923,-177.562,7.929,148.819
C04497=1144.006,249.733,-67.950,-177.560,7.932,148.819
C04498=1144.001,249.981,-67.977,-177.557,7.935,148.819
C04499=1143.997,250.230,-68.005,-177.554,7.938,148.819
C04500=1143.993,250.478,-68.033,-177.551,7.941,148.818
C04501=1143.988,250.727,-68.060,-177.548,7.944,148.818
C04502=1143.983,250.975,-68.088,-177.546,7.946,148.818
C04503=1143.979,251.224,-68.116,-177.543,7.949,148.818
C04504=1143.975,251.472,-68.143,-177.540,7.952,148.818
C04505=1143.970,251.721,-68.170,-177.537,7.955,148.818
C04506=1143.966,251.969,-68.199,-177.535,7.959,148.818
C04507=1143.962,252.218,-68.226,-177.532,7.961,148.818
C04508=1143.957,252.465,-68.253,-177.529,7.964,148.818
C04509=1143.953,252.715,-68.281,-177.527,7.967,148.818
C04510=1143.949,252.963,-68.309,-177.524,7.970,148.818
C04511=1143.944,253.211,-68.337,-177.521,7.973,148.818
C04512=1143.940,253.460,-68.364,-177.518,7.976,148.818
C04513=1143.935,253.708,-68.392,-177.515,7.979,148.818
C04514=1143.932,253.956,-68.420,-177.513,7.982,148.818
C04515=1143.927,254.205,-68.447,-177.510,7.985,148.818
C04516=1143.923,254.453,-68.475,-177.507,7.988,148.818
C04517=1143.918,254.702,-68.504,-177.504,7.991,148.817
C04518=1143.913,254.950,-68.531,-177.502,7.994,148.818
C04519=1143.910,255.199,-68.559,-177.499,7.997,148.818
C04520=1143.905,255.447,-68.587,-177.496,8.000,148.818
C04521=1143.900,255.695,-68.614,-177.494,8.003,148.817
C04522=1143.896,255.944,-68.643,-177.491,8.006,148.817
C04523=1143.892,256.192,-68.670,-177.488,8.009,148.817
C04524=1143.888,256.440,-68.699,-177.485,8.011,148.817
C04525=1143.883,256.689,-68.727,-177.482,8.014,148.817
C04526=1143.879,256.938,-68.754,-177.480,8.017,148.817
C04527=1143.875,257.186,-68.782,-177.477,8.020,148.817
C04528=1143.870,257.434,-68.810,-177.474,8.024,148.817
C04529=1143.866,257.682,-68.839,-177.472,8.026,148.817
C04530=1143.861,257.930,-68.866,-177.469,8.029,148.817
C04531=1143.858,258.179,-68.895,-177.466,8.032,148.817
C04532=1143.853,258.427,-68.923,-177.463,8.035,148.817
C04533=1143.849,258.676,-68.950,-177.461,8.038,148.817
C04534=1143.844,258.924,-68.978,-177.458,8.041,148.817
C04535=1143.840,259.173,-69.007,-177.455,8.044,148.817
C04536=1143.835,259.421,-69.035,-177.453,8.047,148.817
C04537=1143.831,259.670,-69.063,-177.450,8.050,148.817
C04538=1143.826,259.918,-69.091,-177.447,8.053,148.817
C04539=1143.823,260.166,-69.119,-177.444,8.057,148.817
C04540=1143.818,260.414,-69.148,-177.441,8.060,148.817
C04541=1143.814,260.663,-69.176,-177.438,8.063,148.817
C04542=1143.809,260.911,-69.204,-177.436,8.066,148.817
C04543=1143.805,261.185,-69.235,-177.433,8.069,148.817
C04544=1143.800,261.458,-69.267,-177.430,8.073,148.817
C04545=1143.795,261.732,-69.298,-177.427,8.076,148.817
C04546=1143.790,262.005,-69.329,-177.423,8.079,148.817
C04547=1143.786,262.254,-69.357,-177.421,8.082,148.817
C04548=1143.782,262.502,-69.385,-177.418,8.085,148.816
C04549=1143.777,262.751,-69.414,-177.415,8.088,148.816
C04550=1143.774,262.999,-69.443,-177.413,8.091,148.817
C04551=1143.768,263.247,-69.471,-177.410,8.094,148.816
C04552=1143.765,263.495,-69.499,-177.407,8.097,148.816
C04553=1143.760,263.744,-69.528,-177.404,8.100,148.816
C04554=1143.756,263.992,-69.556,-177.402,8.103,148.816
C04555=1143.752,264.240,-69.585,-177.399,8.106,148.816
C04556=1143.747,264.488,-69.613,-177.396,8.109,148.816
C04557=1143.743,264.737,-69.642,-177.394,8.112,148.816
C04558=1143.738,264.985,-69.670,-177.390,8.116,148.816
C04559=1143.734,265.233,-69.699,-177.388,8.119,148.816
C04560=1143.730,265.482,-69.728,-177.385,8.122,148.816
C04561=1143.725,265.730,-69.755,-177.382,8.125,148.816
C04562=1143.721,265.979,-69.784,-177.380,8.128,148.816
C04563=1143.717,266.227,-69.814,-177.377,8.131,148.816
C04564=1143.712,266.475,-69.841,-177.374,8.134,148.816
C04565=1143.708,266.724,-69.870,-177.372,8.137,148.816
C04566=1143.704,266.972,-69.900,-177.369,8.140,148.816
C04567=1143.699,267.220,-69.927,-177.366,8.143,148.816
C04568=1143.695,267.468,-69.957,-177.363,8.147,148.816
C04569=1143.691,267.717,-69.986,-177.360,8.150,148.816
C04570=1143.686,267.965,-70.013,-177.358,8.153,148.816
C04571=1143.682,268.213,-70.043,-177.355,8.156,148.816
C04572=1143.678,268.462,-70.072,-177.352,8.159,148.816
C04573=1143.674,268.710,-70.100,-177.350,8.162,148.816
C04574=1143.669,268.958,-70.129,-177.347,8.165,148.816
C04575=1143.665,269.207,-70.158,-177.344,8.168,148.816
C04576=1143.661,269.455,-70.186,-177.341,8.171,148.816
C04577=1143.657,269.703,-70.215,-177.338,8.175,148.816
C04578=1143.652,269.952,-70.244,-177.336,8.178,148.816
C04579=1143.648,270.200,-70.274,-177.333,8.181,148.816
C04580=1143.644,270.449,-70.302,-177.330,8.184,148.816
C04581=1143.639,270.696,-70.331,-177.328,8.187,148.816
C04582=1143.635,270.944,-70.360,-177.325,8.190,148.816
C04583=1143.631,271.193,-70.389,-177.322,8.193,148.816
C04584=1143.626,271.442,-70.419,-177.319,8.196,148.816
C04585=1143.622,271.689,-70.446,-177.317,8.200,148.816
C04586=1143.618,271.938,-70.476,-177.314,8.203,148.816
C04587=1143.614,272.186,-70.505,-177.311,8.206,148.816
C04588=1143.609,272.435,-70.534,-177.309,8.209,148.816
C04589=1143.604,272.682,-70.563,-177.306,8.212,148.816
C04590=1143.600,272.931,-70.592,-177.303,8.215,148.816
C04591=1143.596,273.179,-70.622,-177.300,8.218,148.816
C04592=1143.592,273.428,-70.650,-177.298,8.221,148.816
C04593=1143.588,273.676,-70.680,-177.295,8.225,148.816
C04594=1143.584,273.924,-70.709,-177.292,8.228,148.816
C04595=1143.579,274.172,-70.738,-177.289,8.231,148.816
C04596=1143.575,274.421,-70.767,-177.287,8.234,148.816
C04597=1143.571,274.669,-70.796,-177.284,8.237,148.816
C04598=1143.566,274.917,-70.826,-177.282,8.240,148.817
C04599=1143.562,275.165,-70.855,-177.278,8.244,148.816
C04600=1143.558,275.414,-70.885,-177.275,8.247,148.816
C04601=1143.554,275.662,-70.914,-177.273,8.250,148.817
C04602=1143.549,275.910,-70.942,-177.270,8.253,148.817
C04603=1143.545,276.158,-70.972,-177.268,8.256,148.816
C04604=1143.540,276.407,-71.001,-177.265,8.259,148.817
C04605=1143.537,276.655,-71.030,-177.262,8.262,148.817
C04606=1143.533,276.903,-71.060,-177.259,8.266,148.817
C04607=1143.529,277.151,-71.089,-177.257,8.269,148.817
C04608=1143.524,277.399,-71.119,-177.254,8.272,148.817
C04609=1143.519,277.648,-71.149,-177.251,8.275,148.817
C04610=1143.515,277.896,-71.178,-177.249,8.278,148.817
C04611=1143.511,278.144,-71.207,-177.246,8.281,148.817
C04612=1143.506,278.392,-71.237,-177.243,8.285,148.817
C04613=1143.502,278.640,-71.266,-177.240,8.288,148.817
C04614=1143.498,278.889,-71.296,-177.238,8.291,148.817
C04615=1143.494,279.137,-71.325,-177.235,8.294,148.817
C04616=1143.490,279.385,-71.354,-177.232,8.297,148.817
C04617=1143.485,279.633,-71.384,-177.229,8.301,148.817
C04618=1143.481,279.882,-71.413,-177.227,8.304,148.817
C04619=1143.477,280.130,-71.443,-177.224,8.307,148.817
C04620=1143.473,280.378,-71.472,-177.222,8.310,148.817
C04621=1143.469,280.626,-71.502,-177.219,8.313,148.817
C04622=1143.464,280.874,-71.532,-177.216,8.316,148.817
C04623=1143.460,281.123,-71.562,-177.213,8.320,148.817
C04624=1143.456,281.371,-71.591,-177.210,8.323,148.817
C04625=1143.452,281.619,-71.621,-177.208,8.327,148.817
C04626=1143.447,281.867,-71.650,-177.205,8.329,148.817
C04627=1143.443,282.115,-71.681,-177.202,8.332,148.817
C04628=1143.439,282.364,-71.710,-177.200,8.336,148.818
C04629=1143.434,282.612,-71.740,-177.197,8.339,148.818
C04630=1143.430,282.860,-71.769,-177.194,8.343,148.818
C04631=1143.426,283.108,-71.800,-177.192,8.346,148.818
C04632=1143.421,283.356,-71.830,-177.189,8.349,148.818
C04633=1143.417,283.605,-71.859,-177.186,8.353,148.818
C04634=1143.413,283.852,-71.889,-177.183,8.356,148.818
C04635=1143.409,284.101,-71.919,-177.181,8.359,148.818
C04636=1143.404,284.349,-71.949,-177.178,8.362,148.818
C04637=1143.400,284.597,-71.979,-177.175,8.366,148.818
C04638=1143.396,284.845,-72.008,-177.172,8.369,148.818
C04639=1143.391,285.094,-72.038,-177.170,8.372,148.818
C04640=1143.387,285.341,-72.069,-177.167,8.375,148.818
C04641=1143.383,285.590,-72.098,-177.164,8.378,148.818
C04642=1143.380,285.838,-72.129,-177.162,8.382,148.818
C04643=1143.375,286.087,-72.159,-177.159,8.385,148.818
C04644=1143.371,286.334,-72.189,-177.156,8.388,148.818
C04645=1143.366,286.583,-72.219,-177.154,8.391,148.818
C04646=1143.362,286.830,-72.249,-177.151,8.395,148.819
C04647=1143.357,287.106,-72.282,-177.148,8.398,148.819
C04648=1143.353,287.382,-72.316,-177.145,8.402,148.819
C04649=1143.348,287.657,-72.348,-177.142,8.406,148.819
C04650=1143.344,287.932,-72.382,-177.139,8.409,148.819
C04651=1143.339,288.180,-72.413,-177.136,8.413,148.819
C04652=1143.335,288.429,-72.442,-177.134,8.416,148.819
C04653=1143.331,288.676,-72.473,-177.131,8.419,148.819
C04654=1143.327,288.926,-72.503,-177.128,8.422,148.819
C04655=1143.323,289.173,-72.533,-177.125,8.426,148.819
C04656=1143.318,289.421,-72.564,-177.123,8.429,148.819
C04657=1143.314,289.669,-72.593,-177.120,8.432,148.819
C04658=1143.309,289.917,-72.624,-177.118,8.436,148.819
C04659=1143.305,290.165,-72.654,-177.114,8.439,148.819
C04660=1143.301,290.414,-72.685,-177.112,8.443,148.820
C04661=1143.297,290.662,-72.715,-177.109,8.446,148.820
C04662=1143.293,290.910,-72.746,-177.107,8.449,148.820
C04663=1143.289,291.158,-72.775,-177.104,8.453,148.820
C04664=1143.284,291.406,-72.806,-177.101,8.456,148.820
C04665=1143.281,291.655,-72.836,-177.098,8.459,148.820
C04666=1143.276,291.902,-72.867,-177.096,8.462,148.820
C04667=1143.272,292.150,-72.897,-177.093,8.466,148.820
C04668=1143.267,292.399,-72.927,-177.090,8.469,148.820
C04669=1143.264,292.647,-72.958,-177.088,8.472,148.820
C04670=1143.259,292.895,-72.989,-177.085,8.475,148.820
C04671=1143.255,293.143,-73.019,-177.082,8.479,148.821
C04672=1143.251,293.391,-73.050,-177.080,8.482,148.821
C04673=1143.247,293.639,-73.081,-177.077,8.485,148.821
C04674=1143.243,293.888,-73.110,-177.074,8.488,148.821
C04675=1143.238,294.136,-73.141,-177.072,8.492,148.821
C04676=1143.233,294.383,-73.172,-177.069,8.496,148.821
C04677=1143.230,294.632,-73.202,-177.066,8.499,148.821
C04678=1143.226,294.880,-73.233,-177.063,8.503,148.821
C04679=1143.222,295.127,-73.263,-177.061,8.506,148.821
C04680=1143.218,295.376,-73.294,-177.058,8.509,148.821
C04681=1143.213,295.624,-73.325,-177.056,8.512,148.821
C04682=1143.209,295.872,-73.355,-177.053,8.516,148.822
C04683=1143.205,296.120,-73.386,-177.050,8.519,148.822
C04684=1143.201,296.368,-73.417,-177.048,8.522,148.822
C04685=1143.196,296.616,-73.448,-177.045,8.526,148.822
C04686=1143.193,296.865,-73.478,-177.042,8.530,148.822
C04687=1143.188,297.113,-73.509,-177.040,8.532,148.822
C04688=1143.183,297.361,-73.540,-177.037,8.536,148.822
C04689=1143.180,297.609,-73.572,-177.034,8.539,148.822
C04690=1143.176,297.856,-73.602,-177.032,8.543,148.822
C04691=1143.171,298.104,-73.633,-177.029,8.546,148.823
C04692=1143.167,298.353,-73.664,-177.026,8.550,148.823
C04693=1143.163,298.601,-73.695,-177.023,8.553,148.823
C04694=1143.159,298.848,-73.725,-177.021,8.556,148.823
C04695=1143.155,299.097,-73.756,-177.018,8.560,148.823
C04696=1143.150,299.344,-73.787,-177.015,8.563,148.823
C04697=1143.146,299.593,-73.819,-177.013,8.567,148.823
C04698=1143.142,299.841,-73.849,-177.010,8.570,148.823
C04699=1143.137,300.089,-73.880,-177.007,8.574,148.823
C04700=1143.134,300.337,-73.911,-177.005,8.577,148.824
C04701=1143.130,300.585,-73.942,-177.002,8.580,148.824
C04702=1143.126,300.833,-73.973,-176.999,8.584,148.824
C04703=1143.121,301.081,-74.005,-176.997,8.587,148.824
C04704=1143.117,301.329,-74.035,-176.994,8.590,148.824
C04705=1143.113,301.577,-74.067,-176.991,8.594,148.824
C04706=1143.108,301.825,-74.098,-176.989,8.597,148.824
C04707=1143.104,302.073,-74.129,-176.986,8.600,148.824
C04708=1143.100,302.321,-74.160,-176.983,8.604,148.824
C04709=1143.096,302.569,-74.192,-176.981,8.608,148.825
C04710=1143.091,302.817,-74.223,-176.978,8.611,148.825
C04711=1143.087,303.065,-74.253,-176.975,8.615,148.825
C04712=1143.084,303.313,-74.285,-176.973,8.618,148.825
C04713=1143.079,303.561,-74.315,-176.971,8.621,148.825
C04714=1143.075,303.809,-74.347,-176.967,8.625,148.825
C04715=1143.071,304.057,-74.378,-176.965,8.628,148.825
C04716=1143.067,304.305,-74.410,-176.963,8.631,148.826
C04717=1143.063,304.553,-74.441,-176.960,8.636,148.826
C04718=1143.059,304.801,-74.472,-176.957,8.638,148.826
C04719=1143.053,305.049,-74.504,-176.954,8.643,148.826
C04720=1143.050,305.297,-74.536,-176.952,8.646,148.826
C04721=1143.045,305.545,-74.566,-176.949,8.649,148.826
C04722=1143.041,305.793,-74.598,-176.946,8.653,148.826
C04723=1143.037,306.041,-74.630,-176.944,8.656,148.826
C04724=1143.033,306.289,-74.661,-176.941,8.659,148.827
C04725=1143.029,306.537,-74.693,-176.938,8.663,148.827
C04726=1143.025,306.785,-74.723,-176.936,8.666,148.827
C04727=1143.021,307.033,-74.755,-176.933,8.670,148.827
C04728=1143.017,307.281,-74.787,-176.930,8.674,148.827
C04729=1143.013,307.529,-74.818,-176.928,8.677,148.827
C04730=1143.008,307.777,-74.849,-176.925,8.680,148.827
C04731=1143.004,308.025,-74.882,-176.922,8.684,148.828
C04732=1142.999,308.273,-74.913,-176.920,8.687,148.828
C04733=1142.996,308.521,-74.944,-176.917,8.691,148.828
C04734=1142.992,308.769,-74.976,-176.915,8.695,148.828
C04735=1142.988,309.016,-75.008,-176.912,8.698,148.828
C04736=1142.984,309.265,-75.039,-176.909,8.702,148.828
C04737=1142.979,309.513,-75.071,-176.907,8.705,148.829
C04738=1142.975,309.761,-75.103,-176.904,8.708,148.829
C04739=1142.971,310.009,-75.135,-176.901,8.712,148.829
C04740=1142.967,310.256,-75.166,-176.899,8.715,148.829
C04741=1142.963,310.504,-75.198,-176.896,8.719,148.829
C04742=1142.958,310.753,-75.230,-176.893,8.722,148.829
C04743=1142.954,311.000,-75.261,-176.891,8.726,148.830
C04744=1142.950,311.248,-75.293,-176.888,8.730,148.830
C04745=1142.947,311.496,-75.325,-176.886,8.733,148.830
C04746=1142.942,311.744,-75.357,-176.883,8.737,148.830
C04747=1142.938,311.992,-75.389,-176.880,8.740,148.830
C04748=1142.934,312.240,-75.421,-176.878,8.743,148.830
C04749=1142.929,312.488,-75.453,-176.875,8.747,148.831
C04750=1142.926,312.736,-75.485,-176.873,8.751,148.831
C04751=1142.921,313.013,-75.520,-176.870,8.755,148.831
C04752=1142.916,313.291,-75.556,-176.867,8.759,148.831
C04753=1142.912,313.569,-75.591,-176.864,8.763,148.831
C04754=1142.906,313.847,-75.627,-176.860,8.767,148.831
C04755=1142.903,314.095,-75.659,-176.858,8.770,148.832
C04756=1142.899,314.343,-75.691,-176.855,8.774,148.832
C04757=1142.894,314.590,-75.724,-176.853,8.777,148.832
C04758=1142.891,314.838,-75.756,-176.850,8.781,148.832
C04759=1142.887,315.086,-75.788,-176.848,8.785,148.832
C04760=1142.882,315.335,-75.820,-176.845,8.788,148.833
C04761=1142.878,315.582,-75.852,-176.842,8.792,148.833
C04762=1142.874,315.830,-75.884,-176.840,8.795,148.833
C04763=1142.870,316.079,-75.916,-176.837,8.799,148.833
C04764=1142.867,316.326,-75.948,-176.834,8.802,148.833
C04765=1142.862,316.574,-75.980,-176.831,8.806,148.833
C04766=1142.858,316.822,-76.012,-176.829,8.810,148.834
C04767=1142.853,317.070,-76.045,-176.827,8.813,148.834
C04768=1142.850,317.317,-76.077,-176.824,8.817,148.834
C04769=1142.846,317.566,-76.110,-176.821,8.820,148.834
C04770=1142.841,317.813,-76.141,-176.818,8.824,148.834
C04771=1142.837,318.061,-76.174,-176.816,8.828,148.835
C04772=1142.833,318.309,-76.206,-176.813,8.832,148.835
C04773=1142.829,318.557,-76.239,-176.811,8.835,148.835
C04774=1142.825,318.805,-76.271,-176.809,8.838,148.835
C04775=1142.821,319.053,-76.304,-176.806,8.842,148.835
C04776=1142.817,319.300,-76.335,-176.803,8.845,148.836
C04777=1142.812,319.549,-76.368,-176.800,8.850,148.836
C04778=1142.809,319.796,-76.400,-176.798,8.853,148.836
C04779=1142.805,320.044,-76.433,-176.795,8.857,148.836
C04780=1142.801,320.292,-76.465,-176.793,8.860,148.836
C04781=1142.797,320.540,-76.498,-176.790,8.864,148.837
C04782=1142.793,320.788,-76.531,-176.788,8.867,148.837
C04783=1142.788,321.035,-76.562,-176.785,8.872,148.837
C04784=1142.784,321.283,-76.595,-176.782,8.875,148.837
C04785=1142.780,321.531,-76.627,-176.780,8.878,148.838
C04786=1142.776,321.779,-76.660,-176.777,8.882,148.838
C04787=1142.772,322.027,-76.693,-176.775,8.885,148.838
C04788=1142.768,322.275,-76.725,-176.772,8.890,148.838
C04789=1142.764,322.523,-76.758,-176.769,8.893,148.838
C04790=1142.760,322.771,-76.791,-176.767,8.897,148.839
C04791=1142.756,323.019,-76.823,-176.764,8.900,148.839
C04792=1142.752,323.266,-76.856,-176.761,8.904,148.839
C04793=1142.748,323.514,-76.889,-176.759,8.907,148.839
C04794=1142.744,323.761,-76.921,-176.756,8.912,148.839
C04795=1142.739,324.009,-76.954,-176.754,8.915,148.840
C04796=1142.735,324.258,-76.986,-176.751,8.919,148.840
C04797=1142.731,324.505,-77.019,-176.748,8.922,148.840
C04798=1142.727,324.753,-77.052,-176.745,8.926,148.840
C04799=1142.723,325.000,-77.085,-176.743,8.929,148.840
C04800=1142.719,325.249,-77.118,-176.740,8.934,148.841
C04801=1142.715,325.496,-77.151,-176.738,8.937,148.841
C04802=1142.711,325.744,-77.183,-176.735,8.941,148.841
C04803=1142.707,325.992,-77.216,-176.733,8.944,148.841
C04804=1142.703,326.240,-77.249,-176.730,8.949,148.842
C04805=1142.699,326.488,-77.282,-176.728,8.952,148.842
C04806=1142.694,326.735,-77.315,-176.725,8.956,148.842
C04807=1142.691,326.983,-77.348,-176.723,8.959,148.842
C04808=1142.687,327.231,-77.380,-176.720,8.963,148.843
C04809=1142.682,327.479,-77.413,-176.717,8.966,148.843
C04810=1142.678,327.727,-77.446,-176.714,8.971,148.843
C04811=1142.674,327.974,-77.480,-176.712,8.974,148.843
C04812=1142.670,328.222,-77.513,-176.710,8.978,148.844
C04813=1142.666,328.470,-77.546,-176.707,8.981,148.844
C04814=1142.663,328.717,-77.578,-176.704,8.986,148.844
C04815=1142.658,328.965,-77.612,-176.702,8.989,148.844
C04816=1142.654,329.213,-77.645,-176.699,8.993,148.844
C04817=1142.650,329.460,-77.678,-176.697,8.996,148.845
C04818=1142.647,329.709,-77.711,-176.694,9.000,148.845
C04819=1142.642,329.957,-77.745,-176.691,9.004,148.845
C04820=1142.638,330.204,-77.778,-176.689,9.008,148.846
C04821=1142.634,330.452,-77.811,-176.687,9.011,148.846
C04822=1142.630,330.700,-77.844,-176.684,9.015,148.846
C04823=1142.626,330.948,-77.877,-176.681,9.019,148.846
C04824=1142.622,331.195,-77.910,-176.678,9.023,148.846
C04825=1142.618,331.443,-77.944,-176.676,9.026,148.847
C04826=1142.613,331.691,-77.977,-176.674,9.030,148.847
C04827=1142.609,331.938,-78.010,-176.671,9.033,148.847
C04828=1142.605,332.186,-78.043,-176.668,9.038,148.847
C04829=1142.602,332.435,-78.077,-176.666,9.041,148.848
C04830=1142.598,332.682,-78.110,-176.663,9.045,148.848
C04831=1142.594,332.929,-78.144,-176.661,9.049,148.848
C04832=1142.590,333.177,-78.177,-176.658,9.053,148.849
C04833=1142.585,333.425,-78.210,-176.655,9.057,148.849
C04834=1142.581,333.673,-78.243,-176.653,9.060,148.849
C04835=1142.577,333.920,-78.276,-176.650,9.064,148.849
C04836=1142.574,334.168,-78.310,-176.648,9.068,148.850
C04837=1142.570,334.416,-78.344,-176.645,9.072,148.850
C04838=1142.565,334.664,-78.377,-176.643,9.075,148.850
C04839=1142.561,334.911,-78.411,-176.640,9.079,148.850
C04840=1142.557,335.159,-78.444,-176.638,9.083,148.851
C04841=1142.553,335.407,-78.478,-176.635,9.087,148.851
C04842=1142.549,335.655,-78.511,-176.632,9.091,148.851
C04843=1142.545,335.902,-78.545,-176.630,9.094,148.851
C04844=1142.541,336.150,-78.578,-176.627,9.098,148.852
C04845=1142.537,336.397,-78.613,-176.625,9.102,148.852
C04846=1142.533,336.646,-78.646,-176.622,9.106,148.852
C04847=1142.529,336.893,-78.679,-176.620,9.109,148.852
C04848=1142.525,337.140,-78.713,-176.617,9.113,148.853
C04849=1142.521,337.388,-78.746,-176.614,9.117,148.853
C04850=1142.518,337.636,-78.781,-176.612,9.121,148.853
C04851=1142.513,337.884,-78.814,-176.609,9.125,148.854
C04852=1142.509,338.131,-78.848,-176.607,9.128,148.854
C04853=1142.505,338.379,-78.881,-176.604,9.132,148.854
C04854=1142.502,338.627,-78.916,-176.602,9.136,148.854
C04855=1142.497,338.907,-78.954,-176.599,9.141,148.855
C04856=1142.492,339.188,-78.993,-176.596,9.145,148.855
C04857=1142.487,339.469,-79.030,-176.593,9.149,148.855
C04858=1142.483,339.749,-79.068,-176.591,9.153,148.856
C04859=1142.479,339.997,-79.103,-176.588,9.158,148.856
C04860=1142.475,340.244,-79.137,-176.585,9.161,148.856
C04861=1142.471,340.492,-79.170,-176.583,9.165,148.857
C04862=1142.467,340.740,-79.205,-176.580,9.169,148.857
C04863=1142.463,340.987,-79.238,-176.578,9.173,148.857
C04864=1142.459,341.235,-79.272,-176.575,9.177,148.858
C04865=1142.455,341.483,-79.306,-176.573,9.180,148.858
C04866=1142.451,341.730,-79.340,-176.570,9.184,148.858
C04867=1142.446,341.978,-79.374,-176.567,9.189,148.859
C04868=1142.443,342.226,-79.408,-176.565,9.192,148.859
C04869=1142.439,342.473,-79.442,-176.562,9.196,148.859
C04870=1142.434,342.721,-79.476,-176.560,9.200,148.859
C04871=1142.431,342.969,-79.510,-176.557,9.204,148.860
C04872=1142.426,343.216,-79.545,-176.554,9.208,148.860
C04873=1142.423,343.463,-79.578,-176.552,9.211,148.860
C04874=1142.419,343.711,-79.613,-176.549,9.215,148.861
C04875=1142.414,343.959,-79.646,-176.546,9.219,148.861
C04876=1142.410,344.207,-79.681,-176.545,9.223,148.861
C04877=1142.407,344.454,-79.715,-176.542,9.227,148.861
C04878=1142.402,344.702,-79.750,-176.540,9.231,148.862
C04879=1142.399,344.950,-79.784,-176.537,9.235,148.862
C04880=1142.394,345.197,-79.818,-176.534,9.239,148.862
C04881=1142.391,345.445,-79.853,-176.532,9.242,148.863
C04882=1142.386,345.692,-79.887,-176.529,9.246,148.863
C04883=1142.383,345.939,-79.921,-176.527,9.251,148.863
C04884=1142.379,346.187,-79.956,-176.524,9.254,148.864
C04885=1142.375,346.434,-79.990,-176.521,9.258,148.864
C04886=1142.371,346.683,-80.024,-176.519,9.262,148.864
C04887=1142.367,346.930,-80.058,-176.516,9.266,148.865
C04888=1142.363,347.178,-80.093,-176.514,9.270,148.865
C04889=1142.358,347.425,-80.128,-176.512,9.274,148.865
C04890=1142.355,347.672,-80.161,-176.509,9.278,148.866
C04891=1142.351,347.921,-80.196,-176.506,9.282,148.866
C04892=1142.347,348.168,-80.230,-176.504,9.286,148.866
C04893=1142.343,348.416,-80.265,-176.501,9.290,148.867
C04894=1142.338,348.663,-80.299,-176.498,9.294,148.867
C04895=1142.335,348.911,-80.334,-176.497,9.297,148.867
C04896=1142.330,349.158,-80.368,-176.494,9.301,148.867
C04897=1142.327,349.407,-80.403,-176.491,9.306,148.868
C04898=1142.323,349.653,-80.438,-176.489,9.309,148.868
C04899=1142.319,349.901,-80.472,-176.486,9.313,148.869
C04900=1142.314,350.149,-80.507,-176.483,9.317,148.869
C04901=1142.311,350.396,-80.541,-176.481,9.321,148.869
C04902=1142.307,350.644,-80.576,-176.479,9.325,148.869
C04903=1142.303,350.891,-80.611,-176.476,9.330,148.870
C04904=1142.300,351.139,-80.645,-176.474,9.333,148.870
C04905=1142.295,351.386,-80.680,-176.471,9.337,148.871
C04906=1142.291,351.635,-80.715,-176.468,9.341,148.871
C04907=1142.287,351.881,-80.750,-176.466,9.345,148.871
C04908=1142.284,352.129,-80.784,-176.463,9.349,148.871
C04909=1142.279,352.377,-80.819,-176.461,9.353,148.872
C04910=1142.275,352.624,-80.854,-176.459,9.357,148.872
C04911=1142.272,352.872,-80.889,-176.456,9.361,148.873
C04912=1142.268,353.119,-80.923,-176.453,9.365,148.873
C04913=1142.264,353.367,-80.958,-176.451,9.369,148.873
C04914=1142.259,353.614,-80.993,-176.448,9.373,148.874
C04915=1142.256,353.862,-81.028,-176.446,9.377,148.874
C04916=1142.252,354.110,-81.063,-176.443,9.380,148.874
C04917=1142.248,354.357,-81.098,-176.441,9.385,148.875
C04918=1142.244,354.605,-81.133,-176.438,9.389,148.875
C04919=1142.240,354.851,-81.168,-176.436,9.392,148.875
C04920=1142.236,355.099,-81.203,-176.434,9.397,148.876
C04921=1142.232,355.347,-81.238,-176.431,9.401,148.876
C04922=1142.228,355.594,-81.273,-176.429,9.404,148.876
C04923=1142.224,355.842,-81.308,-176.426,9.408,148.877
C04924=1142.220,356.090,-81.343,-176.423,9.413,148.877
C04925=1142.216,356.337,-81.378,-176.420,9.417,148.877
C04926=1142.213,356.584,-81.413,-176.419,9.421,148.878
C04927=1142.209,356.832,-81.448,-176.416,9.425,148.878
C04928=1142.205,357.079,-81.483,-176.413,9.429,148.879
C04929=1142.201,357.327,-81.518,-176.411,9.433,148.879
C04930=1142.197,357.575,-81.554,-176.408,9.437,148.879
C04931=1142.194,357.822,-81.589,-176.406,9.441,148.880
C04932=1142.189,358.069,-81.624,-176.403,9.445,148.880
C04933=1142.185,358.317,-81.659,-176.401,9.449,148.880
C04934=1142.182,358.564,-81.695,-176.398,9.453,148.881
C04935=1142.177,358.811,-81.730,-176.395,9.457,148.881
C04936=1142.173,359.059,-81.765,-176.393,9.462,148.881
C04937=1142.170,359.307,-81.800,-176.391,9.465,148.882
C04938=1142.166,359.554,-81.836,-176.388,9.469,148.882
C04939=1142.162,359.801,-81.871,-176.386,9.474,148.883
C04940=1142.158,360.049,-81.906,-176.383,9.478,148.883
C04941=1142.154,360.297,-81.941,-176.381,9.481,148.883
C04942=1142.151,360.544,-81.977,-176.378,9.485,148.884
C04943=1142.146,360.791,-82.012,-176.375,9.490,148.884
C04944=1142.143,361.039,-82.048,-176.372,9.494,148.884
C04945=1142.139,361.286,-82.083,-176.370,9.498,148.885
C04946=1142.135,361.534,-82.119,-176.368,9.502,148.885
C04947=1142.131,361.781,-82.155,-176.365,9.506,148.885
C04948=1142.126,362.029,-82.189,-176.363,9.510,148.886
C04949=1142.123,362.276,-82.225,-176.360,9.514,148.886
C04950=1142.119,362.524,-82.260,-176.357,9.519,148.887
C04951=1142.115,362.771,-82.296,-176.355,9.523,148.887
C04952=1142.112,363.019,-82.331,-176.352,9.527,148.887
C04953=1142.108,363.266,-82.367,-176.350,9.531,148.888
C04954=1142.103,363.513,-82.403,-176.347,9.535,148.888
C04955=1142.099,363.761,-82.438,-176.344,9.539,148.888
C04956=1142.096,364.008,-82.474,-176.342,9.543,148.889
C04957=1142.092,364.255,-82.510,-176.339,9.548,148.889
C04958=1142.089,364.503,-82.546,-176.336,9.552,148.890
C04959=1142.083,364.786,-82.587,-176.333,9.557,148.890
C04960=1142.079,365.070,-82.628,-176.330,9.561,148.890
C04961=1142.075,365.355,-82.668,-176.327,9.566,148.891
C04962=1142.070,365.638,-82.709,-176.324,9.570,148.891
C04963=1142.067,365.885,-82.745,-176.322,9.575,148.892
C04964=1142.063,366.133,-82.781,-176.319,9.579,148.892
C04965=1142.059,366.380,-82.817,-176.316,9.583,148.892
C04966=1142.055,366.628,-82.853,-176.314,9.588,148.893
C04967=1142.050,366.875,-82.888,-176.311,9.592,148.893
C04968=1142.047,367.122,-82.925,-176.308,9.596,148.894
C04969=1142.043,367.369,-82.960,-176.306,9.601,148.894
C04970=1142.039,367.617,-82.996,-176.303,9.605,148.894
C04971=1142.036,367.864,-83.033,-176.300,9.609,148.895
C04972=1142.032,368.111,-83.068,-176.298,9.613,148.895
C04973=1142.028,368.359,-83.104,-176.295,9.617,148.895
C04974=1142.024,368.606,-83.141,-176.293,9.622,148.896
C04975=1142.021,368.854,-83.176,-176.290,9.626,148.896
C04976=1142.016,369.101,-83.212,-176.287,9.630,148.897
C04977=1142.013,369.348,-83.248,-176.285,9.635,148.897
C04978=1142.008,369.596,-83.285,-176.282,9.639,148.898
C04979=1142.005,369.843,-83.321,-176.279,9.643,148.898
C04980=1142.001,370.091,-83.357,-176.277,9.648,148.898
C04981=1141.997,370.338,-83.393,-176.274,9.652,148.899
C04982=1141.994,370.585,-83.429,-176.271,9.656,148.899
C04983=1141.989,370.833,-83.465,-176.269,9.660,148.899
C04984=1141.986,371.080,-83.501,-176.267,9.664,148.900
C04985=1141.981,371.328,-83.537,-176.264,9.668,148.900
C04986=1141.978,371.574,-83.574,-176.261,9.672,148.901
C04987=1141.974,371.822,-83.611,-176.259,9.677,148.901
C04988=1141.970,372.069,-83.646,-176.256,9.681,148.902
C04989=1141.966,372.316,-83.683,-176.254,9.686,148.902
C04990=1141.963,372.564,-83.718,-176.251,9.690,148.902
C04991=1141.959,372.811,-83.755,-176.248,9.694,148.903
C04992=1141.955,373.058,-83.792,-176.246,9.698,148.903
C04993=1141.951,373.306,-83.828,-176.244,9.702,148.904
C04994=1141.947,373.553,-83.865,-176.241,9.706,148.904
C04995=1141.943,373.800,-83.901,-176.239,9.711,148.905
C04996=1141.939,374.048,-83.937,-176.236,9.715,148.905
C04997=1141.936,374.295,-83.974,-176.234,9.720,148.906
C04998=1141.932,374.542,-84.010,-176.232,9.723,148.906
C04999=1141.928,374.790,-84.046,-176.229,9.727,148.906
C05000=1141.924,375.037,-84.083,-176.226,9.732,148.907
C05001=1141.920,375.284,-84.120,-176.225,9.735,148.907
C05002=1141.917,375.531,-84.156,-176.222,9.740,148.908
C05003=1141.913,375.778,-84.193,-176.220,9.744,148.908
C05004=1141.908,376.026,-84.229,-176.218,9.748,148.909
C05005=1141.905,376.273,-84.265,-176.216,9.752,148.909
C05006=1141.901,376.521,-84.303,-176.213,9.757,148.910
C05007=1141.897,376.768,-84.339,-176.211,9.760,148.910
C05008=1141.894,377.015,-84.376,-176.209,9.764,148.911
C05009=1141.890,377.262,-84.412,-176.207,9.768,148.911
C05010=1141.886,377.509,-84.449,-176.205,9.773,148.912
C05011=1141.882,377.757,-84.485,-176.203,9.776,148.912
C05012=1141.878,378.004,-84.522,-176.201,9.780,148.912
C05013=1141.875,378.252,-84.559,-176.199,9.785,148.913
C05014=1141.871,378.499,-84.596,-176.197,9.788,148.914
C05015=1141.867,378.746,-84.632,-176.195,9.792,148.914
C05016=1141.863,378.993,-84.669,-176.193,9.796,148.915
C05017=1141.859,379.240,-84.706,-176.191,9.800,148.915
C05018=1141.855,379.488,-84.743,-176.189,9.804,148.916
C05019=1141.851,379.735,-84.780,-176.187,9.807,148.916
C05020=1141.848,379.982,-84.816,-176.186,9.811,148.917
C05021=1141.844,380.230,-84.853,-176.184,9.815,148.917
C05022=1141.840,380.477,-84.890,-176.182,9.819,148.918
C05023=1141.836,380.725,-84.927,-176.181,9.823,148.918
C05024=1141.832,380.972,-84.964,-176.179,9.826,148.919
C05025=1141.829,381.218,-85.001,-176.178,9.830,148.920
C05026=1141.825,381.465,-85.038,-176.176,9.834,148.920
C05027=1141.821,381.712,-85.075,-176.175,9.837,148.920
C05028=1141.818,381.960,-85.112,-176.173,9.841,148.921
C05029=1141.813,382.208,-85.149,-176.172,9.845,148.922
C05030=1141.809,382.455,-85.186,-176.171,9.848,148.922
C05031=1141.806,382.702,-85.222,-176.170,9.852,148.923
C05032=1141.802,382.950,-85.259,-176.169,9.855,148.924
C05033=1141.799,383.196,-85.297,-176.168,9.858,148.924
C05034=1141.795,383.443,-85.334,-176.167,9.862,148.925
C05035=1141.790,383.690,-85.370,-176.166,9.865,148.925
C05036=1141.787,383.938,-85.408,-176.165,9.868,148.926
C05037=1141.783,384.186,-85.444,-176.164,9.872,148.927
C05038=1141.779,384.432,-85.482,-176.163,9.875,148.927
C05039=1141.776,384.680,-85.519,-176.163,9.878,148.928
C05040=1141.772,384.927,-85.556,-176.162,9.881,148.929
C05041=1141.768,385.174,-85.592,-176.161,9.884,148.929
C05042=1141.764,385.421,-85.630,-176.162,9.887,148.930
C05043=1141.761,385.669,-85.667,-176.161,9.890,148.931
C05044=1141.757,385.916,-85.704,-176.161,9.893,148.931
C05045=1141.753,386.163,-85.741,-176.160,9.896,148.932
C05046=1141.750,386.410,-85.779,-176.160,9.899,148.933
C05047=1141.745,386.657,-85.816,-176.160,9.902,148.933
C05048=1141.741,386.905,-85.853,-176.160,9.904,148.934
C05049=1141.738,387.151,-85.890,-176.159,9.908,148.935
C05050=1141.734,387.399,-85.927,-176.159,9.910,148.936
C05051=1141.731,387.646,-85.964,-176.160,9.913,148.936
C05052=1141.727,387.893,-86.000,-176.160,9.916,148.937
C05053=1141.723,388.140,-86.038,-176.160,9.918,148.938
C05054=1141.719,388.388,-86.075,-176.160,9.921,148.939
C05055=1141.715,388.635,-86.112,-176.160,9.924,148.939
C05056=1141.712,388.882,-86.150,-176.160,9.926,148.940
C05057=1141.708,389.129,-86.187,-176.161,9.929,148.941
C05058=1141.704,389.376,-86.224,-176.161,9.932,148.942
C05059=1141.701,389.624,-86.262,-176.161,9.934,148.942
C05060=1141.697,389.871,-86.299,-176.162,9.936,148.943
C05061=1141.692,390.118,-86.335,-176.162,9.939,148.944
C05062=1141.689,390.365,-86.373,-176.163,9.942,148.945
C05063=1141.684,390.652,-86.416,-176.163,9.944,148.946
C05064=1141.680,390.940,-86.459,-176.164,9.946,148.946
C05065=1141.675,391.226,-86.503,-176.165,9.949,148.947
C05066=1141.672,391.514,-86.545,-176.166,9.953,148.948
C05067=1141.668,391.760,-86.583,-176.166,9.954,148.949
C05068=1141.664,392.008,-86.620,-176.167,9.957,148.950
C05069=1141.660,392.256,-86.657,-176.168,9.959,148.951
C05070=1141.657,392.502,-86.695,-176.168,9.962,148.951
C05071=1141.653,392.750,-86.732,-176.169,9.964,148.952
C05072=1141.649,392.997,-86.769,-176.170,9.966,148.953
C05073=1141.645,393.244,-86.806,-176.171,9.969,148.954
C05074=1141.642,393.492,-86.844,-176.172,9.971,148.955
C05075=1141.638,393.738,-86.881,-176.173,9.973,148.955
C05076=1141.634,393.985,-86.918,-176.174,9.975,148.956
C05077=1141.630,394.233,-86.955,-176.175,9.977,148.957
C05078=1141.626,394.480,-86.993,-176.175,9.980,148.958
C05079=1141.622,394.727,-87.030,-176.176,9.982,148.959
C05080=1141.619,394.975,-87.067,-176.177,9.984,148.960
C05081=1141.615,395.221,-87.104,-176.179,9.986,148.960
C05082=1141.611,395.469,-87.141,-176.180,9.988,148.961
C05083=1141.607,395.715,-87.179,-176.181,9.990,148.962
C05084=1141.604,395.963,-87.216,-176.182,9.992,148.963
C05085=1141.600,396.210,-87.253,-176.183,9.994,148.964
C05086=1141.596,396.457,-87.291,-176.184,9.996,148.965
C05087=1141.592,396.705,-87.328,-176.185,9.998,148.965
C05088=1141.588,396.952,-87.365,-176.186,10.000,148.966
C05089=1141.584,397.199,-87.402,-176.187,10.002,148.967
C05090=1141.581,397.446,-87.439,-176.188,10.004,148.968
C05091=1141.577,397.693,-87.477,-176.189,10.006,148.969
C05092=1141.573,397.940,-87.514,-176.191,10.008,148.970
C05093=1141.570,398.188,-87.551,-176.192,10.011,148.970
C05094=1141.566,398.435,-87.589,-176.193,10.013,148.971
C05095=1141.562,398.682,-87.625,-176.194,10.015,148.972
C05096=1141.558,398.930,-87.663,-176.196,10.016,148.973
C05097=1141.554,399.176,-87.700,-176.197,10.018,148.974
C05098=1141.550,399.424,-87.737,-176.198,10.020,148.975
C05099=1141.547,399.671,-87.775,-176.199,10.022,148.976
C05100=1141.543,399.918,-87.812,-176.200,10.024,148.976
C05101=1141.539,400.165,-87.849,-176.201,10.027,148.977
C05102=1141.536,400.412,-87.887,-176.202,10.029,148.978
C05103=1141.532,400.660,-87.924,-176.204,10.031,148.979
C05104=1141.528,400.906,-87.961,-176.205,10.032,148.980
C05105=1141.524,401.154,-87.998,-176.206,10.034,148.981
C05106=1141.520,401.401,-88.035,-176.207,10.036,148.981
C05107=1141.517,401.648,-88.073,-176.208,10.038,148.982
C05108=1141.513,401.896,-88.110,-176.210,10.040,148.983
C05109=1141.509,402.143,-88.147,-176.211,10.043,148.984
C05110=1141.505,402.389,-88.184,-176.213,10.044,148.985
C05111=1141.501,402.637,-88.221,-176.214,10.046,148.986
C05112=1141.498,402.884,-88.259,-176.215,10.048,148.986
C05113=1141.494,403.131,-88.296,-176.216,10.050,148.987
C05114=1141.490,403.378,-88.333,-176.217,10.052,148.988
C05115=1141.486,403.626,-88.371,-176.218,10.054,148.989
C05116=1141.482,403.873,-88.408,-176.219,10.056,148.990
C05117=1141.478,404.120,-88.445,-176.221,10.057,148.991
C05118=1141.475,404.367,-88.483,-176.222,10.059,148.991
C05119=1141.471,404.614,-88.519,-176.223,10.062,148.992
C05120=1141.467,404.861,-88.557,-176.224,10.064,148.993
C05121=1141.464,405.109,-88.594,-176.226,10.066,148.994
C05122=1141.460,405.356,-88.631,-176.227,10.068,148.995
C05123=1141.456,405.603,-88.669,-176.228,10.070,148.996
C05124=1141.452,405.851,-88.706,-176.229,10.072,148.997
C05125=1141.448,406.098,-88.743,-176.231,10.073,148.997
C05126=1141.444,406.344,-88.780,-176.232,10.075,148.998
C05127=1141.441,406.592,-88.818,-176.233,10.078,148.999
C05128=1141.437,406.839,-88.855,-176.234,10.080,149.000
C05129=1141.433,407.086,-88.892,-176.235,10.082,149.001
C05130=1141.430,407.334,-88.929,-176.236,10.084,149.002
C05131=1141.426,407.580,-88.967,-176.237,10.086,149.002
C05132=1141.422,407.828,-89.004,-176.238,10.088,149.003
C05133=1141.418,408.076,-89.041,-176.239,10.090,149.004
C05134=1141.414,408.322,-89.078,-176.240,10.092,149.005
C05135=1141.410,408.569,-89.115,-176.241,10.094,149.006
C05136=1141.407,408.817,-89.153,-176.242,10.096,149.007
C05137=1141.403,409.064,-89.190,-176.243,10.098,149.007
C05138=1141.399,409.311,-89.227,-176.244,10.100,149.008
C05139=1141.396,409.558,-89.265,-176.245,10.102,149.009
C05140=1141.392,409.805,-89.302,-176.246,10.104,149.010
C05141=1141.388,410.053,-89.339,-176.247,10.106,149.010
C05142=1141.384,410.299,-89.376,-176.249,10.108,149.011
C05143=1141.380,410.547,-89.413,-176.250,10.110,149.012
C05144=1141.377,410.794,-89.451,-176.251,10.112,149.013
C05145=1141.372,411.041,-89.488,-176.252,10.114,149.014
C05146=1141.369,411.289,-89.525,-176.252,10.116,149.014
C05147=1141.365,411.535,-89.563,-176.253,10.119,149.015
C05148=1141.361,411.782,-89.600,-176.254,10.121,149.016
C05149=1141.358,412.030,-89.637,-176.255,10.123,149.017
C05150=1141.354,412.277,-89.674,-176.256,10.125,149.018
C05151=1141.350,412.524,-89.711,-176.257,10.127,149.019
C05152=1141.346,412.771,-89.749,-176.258,10.129,149.019
C05153=1141.342,413.019,-89.786,-176.259,10.131,149.020
C05154=1141.338,413.266,-89.823,-176.259,10.134,149.021
C05155=1141.335,413.513,-89.861,-176.261,10.136,149.022
C05156=1141.331,413.760,-89.898,-176.261,10.138,149.022
C05157=1141.327,414.007,-89.935,-176.262,10.140,149.023
C05158=1141.324,414.255,-89.972,-176.263,10.142,149.024
C05159=1141.320,414.502,-90.009,-176.263,10.145,149.025
C05160=1141.316,414.749,-90.047,-176.264,10.147,149.026
C05161=1141.314,414.996,-90.085,-176.266,10.149,149.026
C05162=1141.312,415.243,-90.121,-176.266,10.150,149.027
C05163=1141.311,415.491,-90.158,-176.267,10.152,149.028
C05164=1141.310,415.737,-90.196,-176.268,10.155,149.029
C05165=1141.311,415.985,-90.232,-176.268,10.157,149.029
C05166=1141.311,416.232,-90.268,-176.269,10.159,149.030
C05167=1141.313,416.500,-90.309,-176.270,10.161,149.031
C05168=1141.316,416.768,-90.348,-176.271,10.164,149.032
C05169=1141.319,417.036,-90.388,-176.272,10.166,149.033
C05170=1141.323,417.303,-90.427,-176.272,10.168,149.033
C05171=1140.903,417.306,-90.477,-176.274,10.179,149.037
C05172=1140.899,417.035,-90.438,-176.273,10.177,149.036
C05173=1140.895,416.764,-90.398,-176.273,10.174,149.035
C05174=1140.893,416.492,-90.357,-176.272,10.172,149.034
C05175=1140.891,416.220,-90.317,-176.271,10.170,149.034
C05176=1140.890,415.973,-90.280,-176.270,10.167,149.033
C05177=1140.890,415.727,-90.244,-176.270,10.166,149.032
C05178=1140.891,415.479,-90.207,-176.269,10.164,149.031
C05179=1140.892,415.232,-90.170,-176.268,10.162,149.030
C05180=1140.893,414.984,-90.132,-176.267,10.160,149.030
C05181=1140.896,414.737,-90.096,-176.267,10.157,149.029
C05182=1140.900,414.490,-90.058,-176.265,10.155,149.028
C05183=1140.903,414.242,-90.021,-176.265,10.153,149.027
C05184=1140.907,413.996,-89.983,-176.264,10.151,149.027
C05185=1140.911,413.749,-89.947,-176.263,10.149,149.026
C05186=1140.914,413.501,-89.909,-176.262,10.146,149.025
C05187=1140.918,413.254,-89.872,-176.262,10.144,149.024
C05188=1140.922,413.007,-89.835,-176.260,10.142,149.023
C05189=1140.925,412.760,-89.797,-176.259,10.140,149.023
C05190=1140.930,412.513,-89.760,-176.258,10.138,149.022
C05191=1140.933,412.266,-89.723,-176.258,10.135,149.021
C05192=1140.937,412.018,-89.685,-176.257,10.134,149.020
C05193=1140.941,411.771,-89.648,-176.256,10.132,149.019
C05194=1140.945,411.524,-89.611,-176.255,10.129,149.019
C05195=1140.948,411.276,-89.574,-176.254,10.127,149.018
C05196=1140.952,411.030,-89.536,-176.253,10.125,149.017
C05197=1140.956,410.783,-89.499,-176.252,10.123,149.016
C05198=1140.960,410.535,-89.462,-176.251,10.121,149.015
C05199=1140.963,410.288,-89.424,-176.250,10.119,149.014
C05200=1140.967,410.041,-89.388,-176.249,10.117,149.014
C05201=1140.971,409.794,-89.350,-176.248,10.115,149.013
C05202=1140.975,409.547,-89.313,-176.247,10.112,149.012
C05203=1140.979,409.299,-89.276,-176.246,10.110,149.011
C05204=1140.982,409.052,-89.238,-176.245,10.108,149.010
C05205=1140.986,408.805,-89.201,-176.244,10.106,149.010
C05206=1140.990,408.558,-89.164,-176.243,10.104,149.009
C05207=1140.993,408.310,-89.126,-176.242,10.102,149.008
C05208=1140.998,408.063,-89.089,-176.241,10.100,149.007
C05209=1141.001,407.817,-89.052,-176.239,10.099,149.006
C05210=1141.005,407.569,-89.015,-176.238,10.097,149.006
C05211=1141.009,407.322,-88.978,-176.237,10.095,149.005
C05212=1141.013,407.075,-88.940,-176.236,10.093,149.004
C05213=1141.016,406.827,-88.903,-176.235,10.091,149.003
C05214=1141.020,406.581,-88.865,-176.234,10.088,149.002
C05215=1141.024,406.333,-88.829,-176.233,10.086,149.001
C05216=1141.028,406.085,-88.791,-176.232,10.084,149.001
C05217=1141.031,405.839,-88.754,-176.230,10.082,149.000
C05218=1141.035,405.592,-88.717,-176.229,10.080,148.999
C05219=1141.039,405.344,-88.679,-176.228,10.078,148.998
C05220=1141.043,405.097,-88.642,-176.227,10.076,148.997
C05221=1141.047,404.850,-88.605,-176.226,10.074,148.996
C05222=1141.050,404.603,-88.567,-176.224,10.072,148.995
C05223=1141.054,404.356,-88.530,-176.223,10.070,148.995
C05224=1141.058,404.109,-88.493,-176.222,10.068,148.994
C05225=1141.061,403.861,-88.456,-176.221,10.066,148.993
C05226=1141.065,403.614,-88.419,-176.220,10.064,148.992
C05227=1141.069,403.367,-88.381,-176.219,10.062,148.991
C05228=1141.073,403.119,-88.344,-176.217,10.060,148.990
C05229=1141.077,402.873,-88.306,-176.216,10.058,148.989
C05230=1141.081,402.626,-88.270,-176.215,10.056,148.989
C05231=1141.084,402.378,-88.232,-176.213,10.054,148.988
C05232=1141.088,402.131,-88.195,-176.212,10.052,148.987
C05233=1141.092,401.884,-88.158,-176.211,10.050,148.986
C05234=1141.095,401.636,-88.121,-176.210,10.048,148.985
C05235=1141.099,401.390,-88.083,-176.209,10.046,148.984
C05236=1141.103,401.142,-88.046,-176.207,10.045,148.984
C05237=1141.107,400.895,-88.008,-176.206,10.042,148.983
C05238=1141.111,400.648,-87.971,-176.205,10.040,148.982
C05239=1141.115,400.401,-87.935,-176.204,10.038,148.981
C05240=1141.119,400.154,-87.897,-176.203,10.036,148.980
C05241=1141.122,399.906,-87.860,-176.202,10.034,148.979
C05242=1141.126,399.660,-87.822,-176.200,10.032,148.979
C05243=1141.130,399.413,-87.785,-176.199,10.031,148.978
C05244=1141.133,399.165,-87.748,-176.198,10.029,148.977
C05245=1141.137,398.918,-87.711,-176.196,10.026,148.976
C05246=1141.141,398.671,-87.674,-176.195,10.024,148.975
C05247=1141.144,398.424,-87.636,-176.194,10.022,148.974
C05248=1141.149,398.176,-87.599,-176.193,10.020,148.973
C05249=1141.153,397.929,-87.562,-176.192,10.018,148.973
C05250=1141.156,397.682,-87.524,-176.191,10.016,148.972
C05251=1141.160,397.435,-87.487,-176.190,10.014,148.971
C05252=1141.164,397.188,-87.450,-176.189,10.012,148.970
C05253=1141.167,396.940,-87.412,-176.188,10.010,148.969
C05254=1141.171,396.693,-87.376,-176.186,10.008,148.968
C05255=1141.175,396.447,-87.338,-176.185,10.006,148.968
C05256=1141.179,396.199,-87.301,-176.184,10.004,148.967
C05257=1141.182,395.952,-87.263,-176.183,10.002,148.966
C05258=1141.186,395.705,-87.226,-176.182,10.000,148.965
C05259=1141.190,395.457,-87.189,-176.181,9.998,148.964
C05260=1141.194,395.210,-87.152,-176.180,9.996,148.963
C05261=1141.198,394.963,-87.115,-176.179,9.993,148.963
C05262=1141.201,394.716,-87.077,-176.178,9.991,148.962
C05263=1141.205,394.469,-87.040,-176.177,9.989,148.961
C05264=1141.209,394.222,-87.003,-176.176,9.987,148.960
C05265=1141.212,393.974,-86.965,-176.175,9.986,148.959
C05266=1141.217,393.727,-86.928,-176.174,9.983,148.959
C05267=1141.221,393.480,-86.891,-176.173,9.981,148.958
C05268=1141.224,393.233,-86.853,-176.172,9.979,148.957
C05269=1141.228,392.986,-86.817,-176.171,9.976,148.956
C05270=1141.232,392.739,-86.779,-176.171,9.974,148.955
C05271=1141.235,392.491,-86.742,-176.170,9.972,148.955
C05272=1141.239,392.244,-86.705,-176.169,9.970,148.954
C05273=1141.243,391.997,-86.667,-176.168,9.967,148.953
C05274=1141.247,391.749,-86.630,-176.168,9.965,148.952
C05275=1141.251,391.502,-86.593,-176.167,9.962,148.951
C05276=1141.255,391.215,-86.549,-176.166,9.960,148.950
C05277=1141.260,390.928,-86.506,-176.166,9.957,148.950
C05278=1141.264,390.641,-86.463,-176.165,9.954,148.949
C05279=1141.268,390.353,-86.420,-176.165,9.952,148.948
C05280=1141.272,390.106,-86.383,-176.163,9.950,148.947
C05281=1141.276,389.860,-86.345,-176.163,9.947,148.946
C05282=1141.279,389.612,-86.308,-176.163,9.944,148.945
C05283=1141.284,389.364,-86.271,-176.163,9.942,148.945
C05284=1141.287,389.118,-86.233,-176.162,9.939,148.944
C05285=1141.291,388.870,-86.196,-176.162,9.937,148.943
C05286=1141.295,388.623,-86.159,-176.162,9.934,148.942
C05287=1141.299,388.376,-86.122,-176.161,9.932,148.942
C05288=1141.302,388.128,-86.085,-176.161,9.929,148.941
C05289=1141.306,387.881,-86.048,-176.161,9.926,148.940
C05290=1141.310,387.635,-86.010,-176.161,9.923,148.939
C05291=1141.313,387.388,-85.974,-176.161,9.920,148.939
C05292=1141.317,387.140,-85.937,-176.161,9.918,148.938
C05293=1141.321,386.893,-85.899,-176.161,9.915,148.937
C05294=1141.325,386.646,-85.862,-176.162,9.912,148.937
C05295=1141.328,386.398,-85.825,-176.161,9.909,148.936
C05296=1141.332,386.152,-85.787,-176.162,9.907,148.935
C05297=1141.336,385.904,-85.751,-176.162,9.904,148.935
C05298=1141.340,385.656,-85.713,-176.162,9.901,148.934
C05299=1141.344,385.409,-85.676,-176.163,9.898,148.933
C05300=1141.348,385.163,-85.639,-176.164,9.895,148.933
C05301=1141.352,384.916,-85.602,-176.164,9.891,148.932
C05302=1141.355,384.668,-85.565,-176.164,9.889,148.931
C05303=1141.359,384.420,-85.528,-176.165,9.886,148.931
C05304=1141.362,384.174,-85.491,-176.166,9.883,148.930
C05305=1141.366,383.926,-85.454,-176.166,9.879,148.929
C05306=1141.370,383.679,-85.417,-176.168,9.875,148.929
C05307=1141.374,383.432,-85.380,-176.169,9.872,148.928
C05308=1141.378,383.185,-85.342,-176.170,9.869,148.928
C05309=1141.381,382.937,-85.305,-176.170,9.866,148.927
C05310=1141.385,382.690,-85.268,-176.172,9.862,148.926
C05311=1141.389,382.443,-85.232,-176.173,9.859,148.926
C05312=1141.393,382.196,-85.195,-176.174,9.855,148.925
C05313=1141.396,381.948,-85.158,-176.175,9.852,148.924
C05314=1141.400,381.701,-85.121,-176.177,9.848,148.924
C05315=1141.404,381.455,-85.084,-176.179,9.845,148.923
C05316=1141.408,381.207,-85.047,-176.179,9.842,148.923
C05317=1141.412,380.959,-85.010,-176.181,9.838,148.922
C05318=1141.416,380.712,-84.973,-176.182,9.834,148.922
C05319=1141.419,380.465,-84.936,-176.184,9.830,148.921
C05320=1141.423,380.218,-84.900,-176.186,9.826,148.921
C05321=1141.427,379.971,-84.863,-176.187,9.822,148.920
C05322=1141.431,379.723,-84.825,-176.189,9.819,148.920
C05323=1141.435,379.476,-84.789,-176.191,9.815,148.919
C05324=1141.438,379.229,-84.752,-176.193,9.811,148.919
C05325=1141.442,378.982,-84.715,-176.195,9.807,148.918
C05326=1141.447,378.735,-84.679,-176.197,9.803,148.918
C05327=1141.450,378.487,-84.641,-176.199,9.800,148.917
C05328=1141.453,378.240,-84.605,-176.200,9.796,148.916
C05329=1141.457,377.993,-84.568,-176.203,9.791,148.916
C05330=1141.462,377.746,-84.531,-176.205,9.788,148.916
C05331=1141.466,377.498,-84.495,-176.207,9.783,148.915
C05332=1141.469,377.251,-84.458,-176.209,9.780,148.915
C05333=1141.473,377.004,-84.421,-176.211,9.775,148.914
C05334=1141.477,376.756,-84.384,-176.213,9.772,148.914
C05335=1141.480,376.510,-84.348,-176.216,9.767,148.913
C05336=1141.484,376.262,-84.312,-176.218,9.764,148.913
C05337=1141.488,376.014,-84.275,-176.220,9.759,148.912
C05338=1141.492,375.768,-84.239,-176.222,9.755,148.912
C05339=1141.496,375.520,-84.202,-176.224,9.751,148.911
C05340=1141.500,375.273,-84.165,-176.227,9.747,148.911
C05341=1141.503,375.025,-84.129,-176.229,9.743,148.910
C05342=1141.507,374.778,-84.092,-176.231,9.739,148.910
C05343=1141.511,374.531,-84.055,-176.234,9.735,148.910
C05344=1141.515,374.284,-84.019,-176.237,9.730,148.909
C05345=1141.519,374.036,-83.983,-176.238,9.727,148.909
C05346=1141.522,373.789,-83.947,-176.241,9.722,148.908
C05347=1141.526,373.542,-83.910,-176.243,9.718,148.908
C05348=1141.530,373.295,-83.874,-176.246,9.713,148.907
C05349=1141.534,373.047,-83.837,-176.249,9.709,148.907
C05350=1141.538,372.800,-83.801,-176.251,9.705,148.906
C05351=1141.542,372.553,-83.765,-176.253,9.701,148.906
C05352=1141.545,372.305,-83.728,-176.256,9.697,148.906
C05353=1141.549,372.058,-83.692,-176.258,9.693,148.905
C05354=1141.553,371.810,-83.655,-176.261,9.688,148.905
C05355=1141.557,371.563,-83.619,-176.263,9.684,148.904
C05356=1141.561,371.315,-83.583,-176.266,9.680,148.904
C05357=1141.564,371.068,-83.547,-176.269,9.675,148.904
C05358=1141.569,370.821,-83.511,-176.271,9.671,148.903
C05359=1141.572,370.574,-83.474,-176.274,9.667,148.903
C05360=1141.577,370.326,-83.438,-176.277,9.663,148.902
C05361=1141.580,370.079,-83.402,-176.279,9.658,148.902
C05362=1141.584,369.831,-83.366,-176.282,9.654,148.901
C05363=1141.588,369.584,-83.329,-176.285,9.650,148.901
C05364=1141.591,369.337,-83.294,-176.287,9.645,148.901
C05365=1141.595,369.090,-83.257,-176.289,9.642,148.900
C05366=1141.599,368.842,-83.222,-176.292,9.638,148.900
C05367=1141.603,368.594,-83.185,-176.295,9.633,148.900
C05368=1141.607,368.347,-83.149,-176.297,9.629,148.899
C05369=1141.610,368.100,-83.114,-176.300,9.625,148.899
C05370=1141.615,367.853,-83.078,-176.303,9.621,148.898
C05371=1141.619,367.606,-83.042,-176.305,9.616,148.898
C05372=1141.622,367.358,-83.006,-176.308,9.612,148.898
C05373=1141.627,367.111,-82.970,-176.311,9.608,148.897
C05374=1141.630,366.864,-82.934,-176.313,9.603,148.897
C05375=1141.634,366.616,-82.898,-176.316,9.599,148.896
C05376=1141.638,366.368,-82.862,-176.319,9.595,148.896
C05377=1141.642,366.121,-82.826,-176.321,9.590,148.895
C05378=1141.645,365.874,-82.790,-176.324,9.586,148.895
C05379=1141.650,365.626,-82.754,-176.326,9.582,148.895
C05380=1141.654,365.343,-82.713,-176.330,9.577,148.894
C05381=1141.659,365.059,-82.672,-176.332,9.573,148.894
C05382=1141.662,364.775,-82.631,-176.336,9.568,148.893
C05383=1141.667,364.492,-82.590,-176.339,9.562,148.893
C05384=1141.671,364.244,-82.554,-176.341,9.559,148.893
C05385=1141.675,363.997,-82.519,-176.344,9.555,148.892
C05386=1141.679,363.749,-82.483,-176.346,9.551,148.892
C05387=1141.683,363.502,-82.448,-176.349,9.546,148.892
C05388=1141.686,363.255,-82.412,-176.351,9.542,148.891
C05389=1141.691,363.007,-82.376,-176.354,9.538,148.891
C05390=1141.695,362.760,-82.341,-176.357,9.533,148.890
C05391=1141.698,362.512,-82.305,-176.360,9.529,148.890
C05392=1141.702,362.265,-82.270,-176.362,9.525,148.890
C05393=1141.706,362.018,-82.235,-176.364,9.521,148.889
C05394=1141.710,361.770,-82.199,-176.367,9.517,148.889
C05395=1141.713,361.523,-82.163,-176.370,9.513,148.889
C05396=1141.717,361.275,-82.128,-176.373,9.509,148.888
C05397=1141.722,361.027,-82.092,-176.375,9.504,148.888
C05398=1141.726,360.780,-82.057,-176.378,9.500,148.887
C05399=1141.730,360.533,-82.022,-176.380,9.497,148.887
C05400=1141.733,360.285,-81.986,-176.383,9.492,148.887
C05401=1141.737,360.038,-81.951,-176.385,9.488,148.886
C05402=1141.741,359.791,-81.915,-176.388,9.484,148.886
C05403=1141.745,359.543,-81.880,-176.390,9.480,148.885
C05404=1141.749,359.295,-81.845,-176.393,9.476,148.885
C05405=1141.753,359.048,-81.809,-176.395,9.472,148.885
C05406=1141.757,358.801,-81.774,-176.398,9.468,148.885
C05407=1141.761,358.553,-81.739,-176.401,9.463,148.884
C05408=1141.765,358.305,-81.704,-176.403,9.460,148.884
C05409=1141.768,358.058,-81.668,-176.406,9.456,148.883
C05410=1141.772,357.811,-81.633,-176.408,9.451,148.883
C05411=1141.776,357.563,-81.598,-176.411,9.447,148.883
C05412=1141.780,357.315,-81.563,-176.413,9.444,148.882
C05413=1141.784,357.068,-81.528,-176.415,9.439,148.882
C05414=1141.788,356.820,-81.493,-176.418,9.435,148.882
C05415=1141.792,356.573,-81.457,-176.420,9.432,148.881
C05416=1141.796,356.325,-81.422,-176.423,9.428,148.881
C05417=1141.799,356.078,-81.388,-176.426,9.423,148.880
C05418=1141.803,355.831,-81.352,-176.428,9.419,148.880
C05419=1141.807,355.583,-81.317,-176.431,9.416,148.880
C05420=1141.811,355.336,-81.282,-176.433,9.411,148.879
C05421=1141.815,355.088,-81.247,-176.436,9.407,148.879
C05422=1141.820,354.841,-81.212,-176.438,9.404,148.879
C05423=1141.823,354.593,-81.177,-176.441,9.400,148.878
C05424=1141.827,354.345,-81.142,-176.443,9.395,148.878
C05425=1141.831,354.098,-81.108,-176.445,9.392,148.878
C05426=1141.835,353.851,-81.072,-176.448,9.387,148.877
C05427=1141.839,353.603,-81.038,-176.451,9.383,148.877
C05428=1141.843,353.356,-81.002,-176.454,9.379,148.877
C05429=1141.847,353.108,-80.968,-176.456,9.375,148.876
C05430=1141.850,352.861,-80.933,-176.458,9.371,148.876
C05431=1141.854,352.613,-80.898,-176.461,9.367,148.875
C05432=1141.858,352.365,-80.863,-176.463,9.364,148.875
C05433=1141.863,352.118,-80.828,-176.466,9.359,148.875
C05434=1141.867,351.870,-80.793,-176.469,9.355,148.875
C05435=1141.870,351.623,-80.759,-176.471,9.352,148.874
C05436=1141.874,351.375,-80.724,-176.474,9.348,148.874
C05437=1141.879,351.128,-80.689,-176.476,9.343,148.873
C05438=1141.883,350.880,-80.655,-176.478,9.340,148.873
C05439=1141.886,350.632,-80.620,-176.481,9.336,148.873
C05440=1141.890,350.385,-80.585,-176.484,9.332,148.873
C05441=1141.894,350.137,-80.550,-176.486,9.328,148.872
C05442=1141.898,349.890,-80.517,-176.489,9.324,148.872
C05443=1141.902,349.642,-80.482,-176.491,9.319,148.871
C05444=1141.906,349.395,-80.447,-176.493,9.316,148.871
C05445=1141.909,349.147,-80.412,-176.496,9.312,148.871
C05446=1141.914,348.900,-80.378,-176.499,9.308,148.871
C05447=1141.918,348.652,-80.343,-176.501,9.304,148.870
C05448=1141.922,348.405,-80.309,-176.504,9.300,148.870
C05449=1141.926,348.156,-80.274,-176.506,9.296,148.869
C05450=1141.930,347.909,-80.240,-176.509,9.292,148.869
C05451=1141.934,347.661,-80.206,-176.511,9.288,148.869
C05452=1141.938,347.414,-80.171,-176.514,9.284,148.869
C05453=1141.941,347.166,-80.137,-176.516,9.281,148.868
C05454=1141.946,346.919,-80.102,-176.519,9.276,148.868
C05455=1141.950,346.672,-80.067,-176.522,9.272,148.868
C05456=1141.953,346.424,-80.033,-176.524,9.269,148.867
C05457=1141.958,346.177,-79.999,-176.527,9.265,148.867
C05458=1141.961,345.929,-79.964,-176.529,9.261,148.867
C05459=1141.966,345.681,-79.931,-176.531,9.257,148.866
C05460=1141.969,345.433,-79.896,-176.534,9.253,148.866
C05461=1141.974,345.186,-79.862,-176.536,9.249,148.866
C05462=1141.978,344.938,-79.828,-176.539,9.245,148.865
C05463=1141.982,344.690,-79.793,-176.542,9.241,148.865
C05464=1141.986,344.443,-79.759,-176.544,9.238,148.865
C05465=1141.989,344.195,-79.724,-176.547,9.233,148.865
C05466=1141.993,343.948,-79.691,-176.549,9.229,148.864
C05467=1141.998,343.701,-79.656,-176.552,9.226,148.864
C05468=1142.001,343.452,-79.623,-176.554,9.221,148.863
C05469=1142.006,343.205,-79.588,-176.557,9.218,148.863
C05470=1142.009,342.957,-79.554,-176.560,9.214,148.863
C05471=1142.014,342.709,-79.519,-176.562,9.210,148.863
C05472=1142.018,342.462,-79.486,-176.564,9.206,148.862
C05473=1142.021,342.214,-79.452,-176.567,9.202,148.862
C05474=1142.026,341.966,-79.418,-176.570,9.198,148.862
